// The data values inludes 17 bytes, which can be dynamically allocated as needed for each data field based on the size of the number

// Group Input mapping on robot appears as follows

// giKey1 : USINT;               giData1 : USINT;

// giKey2 : USINT;               giData2 : USINT;

// giKey3 : USINT;               giData3 : USINT;

// giKey4 : USINT;               giData4 : USINT;

// giKey5 : USINT;               giData5 : USINT;

// giKey6 : USINT;               giData6 : USINT;

// ...                           ...

// Example:

// Wall SAM ID is the first field of WallInfo step which is a large number 157864127 with needing 4 bytes to send.

// The next field of WallInfo is wall length which is 2000mm requiring 2 bytes to send.

// giKey1 is set to 4 and the number is divided into bytes occupying giData1,giData2,giData3, and giData4.

// giKey2 is set to 2 and the number is divided into bytes occupying giData5 and giData6.

// Function to pack NumbersToSend into bytes and determine key values

// first clear array

FOR i := 0 TO 14 DO
    Recipe_ByteQtyKey[i] := 0;
END_FOR

FOR i := 0 TO 16 DO
    Recipe_PackedBytes[i] := 0;
END_FOR

index := 0;

FOR i := 0 TO 10 DO

    // Determine how many bytes each number will occupy

    Recipe_ByteQtyKey[i] := 1;

    FOR j := 1 TO 3 DO
        IF ABS(RecipeData_ToSend[i]) > EXPT(2, (8 * j) - 1) THEN
            Recipe_ByteQtyKey[i] := INT_TO_USINT(j) + 1;

            // Make it easier to unpack by forcing data to be USINT (1), UINT (2) or UDINT (4)

            IF Recipe_ByteQtyKey[i] = 3 THEN
                Recipe_ByteQtyKey[i] := 4;
            END_IF
        END_IF
    END_FOR

    // Handle signed numbers

    numberToPack := RecipeData_ToSend[i];

    IF numberToPack < 0 THEN
        // Convert to Two's Complement for the required byte size

        CASE Recipe_ByteQtyKey[i] OF
            1:
                numberToPack := numberToPack AND 16#FF; // Mask for 8 bits
            2:
                numberToPack := numberToPack AND 16#FFFF; // Mask for 16 bits
            4:
                numberToPack := numberToPack AND 16#FFFFFFFF; // Mask for 32 bits
        END_CASE;
    END_IF

    // Now extract individual bytes from signed number

    IF Recipe_ByteQtyKey[i] = 1 THEN
        Recipe_PackedBytes[index] := UDINT_TO_USINT(numberToPack);
        index                     := index + 1;
    ELSE
        FOR j := Recipe_ByteQtyKey[i] - 1 TO 1 BY -1 DO
            Recipe_PackedBytes[index] := UDINT_TO_USINT(SHR(numberToPack, 8 * j));
            index                     := index + 1;
        END_FOR

        // Get the last byte

        Recipe_PackedBytes[index] := UDINT_TO_USINT(numberToPack);
        index                     := index + 1;
    END_IF

END_FOR;
END_METHOD

PROPERTY OtherInputs : ARRAY[0..7] OF USINT
GET
PUBLIC
VAR
END_VAR
OtherInputs := OtherInputsArray;
END_GET
END_PROPERTY

PROPERTY OtherOutputs : ARRAY[0..7] OF USINT
SET
PUBLIC
VAR
END_VAR
OtherOutputsArray := OtherOutputs;
END_SET
END_PROPERTY

END_FUNCTION_BLOCK

// Machine/Components/Safety/FB_Component_Safety
FUNCTION_BLOCK FB_Component_Safety EXTENDS FB_ComponentBase_SR
VAR_INPUT
    _SystemState : Tc3_PackML_V2.E_PMLState;
END_VAR

VAR_OUTPUT
END_VAR

VAR CONSTANT
    MAX_MGB_DOORS               : UDINT := 7;
    MAX_ESTOPS                  : UDINT := 8;
    MAX_LIGHT_CURTAINS          : UDINT := 4;
    MAX_AREA_SCANNERS           : UDINT := 3;
    COMPONENT_ALARM_COUNT       : UINT  := 9;
    MAX_PREPLATE_DOORS          : UDINT := 5;
    MAX_PREPLATE_LIGHT_CURTAINS : UDINT := 3;
END_VAR

VAR
    //Alarming
    ComponentAlarms : ARRAY[1..COMPONENT_ALARM_COUNT] OF FB_TcAlarm;

    // Component definitions here
    MGB_Door                      : ARRAY[1..MAX_MGB_DOORS] OF FB_Component_MGB_Door;
    E_Stop                        : ARRAY[1..MAX_ESTOPS] OF FB_DualChannelMonitor;
    E_Stop_Status                 : ARRAY[1..MAX_ESTOPS] OF ST_DualChannel_HMIStatus;
    Light_Curtains                : ARRAY[1..MAX_LIGHT_CURTAINS] OF FB_DualChannelMonitor;
    Light_Curtain_Status          : ARRAY[1..MAX_LIGHT_CURTAINS] OF ST_DualChannel_HMIStatus;
    Area_Scanners                 : ARRAY[1..MAX_AREA_SCANNERS] OF FB_DigitalSensor;
    Preplate_Doors                : ARRAY[1..MAX_PREPLATE_DOORS] OF FB_DualChannelMonitor;
    Preplate_Door_Status          : ARRAY[1..MAX_PREPLATE_DOORS] OF ST_DualChannel_HMIStatus;
    Light_Curtains_Preplate       : ARRAY[1..MAX_PREPLATE_LIGHT_CURTAINS] OF FB_DualChannelMonitor;
    Light_Curtain_Preplate_Status : ARRAY[1..MAX_PREPLATE_LIGHT_CURTAINS] OF ST_DualChannel_HMIStatus;

    FlashingLight : FB_PulseGenerator;

    SafetyRUN     AT %Q* : BOOL := TRUE;
    SafetyErrAckn AT %Q* : BOOL;
    SafetyReset   AT %Q* : BOOL;

    SafetyIsReset AT %I* : BOOL;
    SS1Input      AT %I* : BIT;
    SS1Output     AT %Q* : BIT;

    AirPressureOK AT %I* : BOOL;

    PrePlateAirPressureOK AT %I* : BOOL;

    OutfeedSafetyReset AT %Q* : BOOL;

    OutfeedSafetyIsReset AT %I* : BOOL;

    AutostopIsReset AT %I* : BOOL;

    OutfeedSafetyReset_Button3 AT %I* : BOOL;

    OutfeedSafetyReset_Button2 AT %I* : BOOL;

    OutfeedSafetyReset_HMI AT %I* : BOOL;

    SafetyStop AT %Q* : BOOL;

    SafetyOK_HMI_STATE : USINT;

    AutoStopOK_HMI_STATE : USINT;

    OutfeedAutoStopOK_HMI_STATE : USINT;

    SafetyOK_HMI_TEXT : STRING;

    AutoStopOK_HMI_TEXT : STRING;

    OutfeedAutoStopOK_HMI_TEXT : STRING;

    safetyState                   : USINT;
    tempSafetyOK_Main             : BOOL;
    tempSafetyCanBeReset_Main     : BOOL;
    tempSafetyReset_Main          : BOOL;
    tempSafetyOK_AutoStop         : BOOL;
    tempSafetyCanBeReset_AutoStop : BOOL;
    tempSafetyReset_AutoStop      : BOOL;
    tempSafetyOK_Outfeed          : BOOL;
    tempSafetyCanBeReset_Outfeed  : BOOL;
    tempSafetyReset_Outfeed       : BOOL;
    MainSafetyCanBeReset          : BOOL;
    AutoStopSafetyCanBeReset      : BOOL;
    OutfeedSafetyCanBeReset       : BOOL;
END_VAR

//! @summary This method serves as the entry point for all underlying FB logic
METHOD PUBLIC CyclicLogic

//! @description This method should be called cyclically by descendant function blocks by invoking <c>SUPER^.CyclicLogic()</c>.  Alternatively, the contents of this method could be reimplemented entirely in which case a call to this method would not be necessary.
// MGB_Door Names

MGB_Door[1].Name := 'Infeed';
MGB_Door[2].Name := 'Pre-Press';
MGB_Door[3].Name := 'Post_Press';
MGB_Door[4].Name := 'Assembly';
MGB_Door[5].Name := 'Jig_3 Door';
MGB_Door[6].Name := 'Jig_2 Door';
MGB_Door[7].Name := 'Preplate Cell'; // Button box and estop combined into "MGB Door" 

//Estop names
E_Stop[1].Name := 'MBI 1';
E_Stop[2].Name := 'MBI 1 Cable';
E_Stop[3].Name := 'MBI 2';
E_Stop[4].Name := 'MBI 2 Cable';
E_Stop[5].Name := 'HMI';
E_Stop[6].Name := 'Jig 3 Pendant';
E_Stop[7].Name := 'Jig 2 Pendant';
E_Stop[8].Name := 'Roof Truss Core';

//Outfeed Light curtain names
Light_Curtains[1].Name := 'Curtain 1';
Light_Curtains[2].Name := 'Curtain 2';
Light_Curtains[3].Name := 'Curtain 3';
Light_Curtains[4].Name := 'Curtain 4';

//Preplate Light curtain names
Light_Curtains_Preplate[1].Name := 'Curtain 1';
Light_Curtains_Preplate[2].Name := 'Curtain 2';
Light_Curtains_Preplate[3].Name := 'Curtain 3';

//Outfeed Light curtain names
Preplate_Doors[1].Name := 'Rack 1';
Preplate_Doors[2].Name := 'Rack 2';
Preplate_Doors[3].Name := 'Rack 3';
Preplate_Doors[4].Name := 'Rack 4';
Preplate_Doors[5].Name := 'Rack 5';

HMI_Status_Estops();
HMI_Status_LightCurtains();
HMI_Status_Preplate();

FOR i := 1 TO MAX_PREPLATE_DOORS DO
    Preplate_Doors[i].CyclicLogic();
    Preplate_Doors[i].InSimulation := _Simulate;
END_FOR

FOR i := 1 TO MAX_PREPLATE_LIGHT_CURTAINS DO
    Light_Curtains_Preplate[i].CyclicLogic();
    Light_Curtains_Preplate[i].InSimulation := _Simulate;
END_FOR

// Initialise Component

FlashingLight.OffTime := T#500MS;
FlashingLight.OnTime  := T#500MS;

FlashingLight.CyclicLogic();

MainSafetyCanBeReset := TRUE;

FOR i := 1 TO MAX_ESTOPS DO
    MainSafetyCanBeReset := MainSafetyCanBeReset AND E_Stop[i].BothChannelsOK;
END_FOR

FOR i := 1 TO MAX_MGB_DOORS DO
    MainSafetyCanBeReset := MainSafetyCanBeReset AND MGB_Door[i].Estop_CH_OK;
END_FOR

HMI_Indicators(Area             := 'Main',
               HMI_Text         := SafetyOK_HMI_TEXT,
               HMI_State        := SafetyOK_HMI_STATE,
               SafetyOK         := SafetyIsReset OR (_Simulate AND tempSafetyOK_Main),
               SafetyCanBeReset := MainSafetyCanBeReset,
               SafetyReset      := SafetyReset OR (tempSafetyReset_Main AND _Simulate));

IF MainSafetyCanBeReset AND _Simulate AND SafetyReset THEN
    tempSafetyOK_Main := TRUE;
ELSIF MainSafetyCanBeReset = FALSE THEN
    tempSafetyOK_Main := FALSE;
END_IF

AutoStopSafetyCanBeReset := TRUE;

FOR i := 1 TO MAX_MGB_DOORS - 2 DO
    AutoStopSafetyCanBeReset := AutoStopSafetyCanBeReset AND MGB_Door[i].AutoStop_CH_OK;
END_FOR

AutoStopSafetyCanBeReset := MainSafetyCanBeReset AND AutoStopSafetyCanBeReset;

HMI_Indicators(Area             := 'AutoStop',
               HMI_Text         := AutoStopOK_HMI_TEXT,
               HMI_State        := AutoStopOK_HMI_STATE,
               SafetyOK         := (AutostopIsReset AND SafetyIsReset) OR (_Simulate AND tempSafetyOK_AutoStop),
               SafetyCanBeReset := AutoStopSafetyCanBeReset,
               SafetyReset      := FALSE);

IF AutoStopSafetyCanBeReset AND _Simulate THEN
    tempSafetyOK_AutoStop := TRUE;
ELSIF AutoStopSafetyCanBeReset = FALSE THEN
    tempSafetyOK_AutoStop := FALSE;
END_IF

OutfeedSafetyCanBeReset := TRUE;

FOR i := 1 TO MAX_LIGHT_CURTAINS DO
    OutfeedSafetyCanBeReset := Light_Curtains[i].BothChannelsOK AND OutfeedSafetyCanBeReset;
END_FOR

OutfeedSafetyCanBeReset := MGB_Door[5].AutoStop_CH_OK AND OutfeedSafetyCanBeReset;
OutfeedSafetyCanBeReset := MGB_Door[6].AutoStop_CH_OK AND OutfeedSafetyCanBeReset;
OutfeedSafetyCanBeReset := MainSafetyCanBeReset AND OutfeedSafetyCanBeReset;

HMI_Indicators(Area             := 'Outfeed',
               HMI_Text         := OutfeedAutoStopOK_HMI_TEXT,
               HMI_State        := OutfeedAutoStopOK_HMI_STATE,
               SafetyOK         := (OutfeedSafetyIsReset AND SafetyIsReset) OR (_Simulate AND tempSafetyOK_Outfeed),
               SafetyCanBeReset := OutfeedSafetyCanBeReset,
               SafetyReset      := OutfeedSafetyReset OR (tempSafetyReset_Outfeed AND _Simulate));

IF OutfeedSafetyCanBeReset AND _Simulate AND OutfeedSafetyReset THEN
    tempSafetyOK_Outfeed := TRUE;
ELSIF OutfeedSafetyCanBeReset = FALSE THEN
    tempSafetyOK_Outfeed := FALSE;
END_IF

SS1Output := NOT SS1Input;

IF NOT _InitComplete THEN
    _InitComplete := Initialize();
    RETURN;
END_IF

IF SafetyReset THEN
    SafetyErrAckn := TRUE;
ELSE
    SafetyErrAckn := FALSE;
END_IF

OutfeedSafetyReset := OutfeedSafetyReset_Button3 OR OutfeedSafetyReset_Button2 OR OutfeedSafetyReset_HMI;

FOR i := 1 TO MAX_MGB_DOORS DO

    MGB_Door[i].CyclicLogic();
    MGB_Door[i].InSimulation := _Simulate;

    //Button lights and lock

    CASE _SystemState OF
        ePMLState_Idle:
            MGB_Door[i].Pause_LED.TurnOff();
            MGB_Door[i].Resume_LED.Flash();
            MGB_Door[i].Lock_Door.TurnOff();
        ePMLState_Holding, ePMLState_Suspending:
            MGB_Door[i].Pause_LED.Flash();
            MGB_Door[i].Resume_LED.TurnOff();
            MGB_Door[i].Lock_Door.TurnOn();
        ePMLState_Held, ePMLState_Suspended:
            MGB_Door[i].Pause_LED.TurnOff();
            MGB_Door[i].Resume_LED.TurnOn();
            MGB_Door[i].Lock_Door.TurnOff();
        ePMLState_Starting, ePMLState_Unholding, ePMLState_Unsuspending:
            MGB_Door[i].Pause_LED.TurnOff();
            MGB_Door[i].Resume_LED.Flash();
            MGB_Door[i].Lock_Door.TurnOn();
        ePMLState_Execute:
            MGB_Door[i].Pause_LED.TurnOn();
            MGB_Door[i].Resume_LED.TurnOff();
            MGB_Door[i].Lock_Door.TurnOn();
    ELSE
        MGB_Door[i].Pause_LED.TurnOff();
        MGB_Door[i].Resume_LED.TurnOff();
        MGB_Door[i].Lock_Door.TurnOff();
    END_CASE

    //estop light

    IF SafetyIsReset THEN
        MGB_Door[i].Estop_LED.TurnOff();
    ELSE
        IF MGB_Door[i].Estop_CH_OK THEN
            MGB_Door[i].Estop_LED.Flash();
        ELSE
            MGB_Door[i].Estop_LED.TurnOn();
        END_IF
        MGB_Door[i].Lock_Door.TurnOff();
    END_IF
    MGB_Door[i].SafetyReset := SafetyReset;
END_FOR

FOR i := 1 TO MAX_ESTOPS DO
    E_Stop[i].CyclicLogic();
    E_Stop[i].InSimulation := _Simulate;

    IF SafetyIsReset THEN
        E_Stop[i].LED.TurnOff();
    ELSE
        IF E_Stop[i].BothChannelsOK THEN
            E_Stop[i].LED.Flash();
        ELSE
            E_Stop[i].LED.TurnOn();
        END_IF
    END_IF
END_FOR

FOR i := 1 TO MAX_LIGHT_CURTAINS DO
    Light_Curtains[i].CyclicLogic();
    Light_Curtains[i].InSimulation := _Simulate;
END_FOR

SafetyStop := NOT (SafetyIsReset) OR NOT (AutostopIsReset);

SUPER^.CyclicLogic();
END_METHOD

(*! @summary Initializes event function blocks using this components's name*)
METHOD PROTECTED CreateEvents
F_CreateAllEventsInClass(Alarms     := ComponentAlarms,
                         ClassSize  := SIZEOF(TC_EVENTS.AMDTruss),
                         pInitEvent := ADR(TC_EVENTS.AMDTruss.InitReferenceEvent),
                         Prefix     := _Name);
END_METHOD

METHOD HMI_Indicators

VAR_INPUT
    Area             : STRING;
    HMI_Text         : REFERENCE TO STRING;
    HMI_State        : REFERENCE TO USINT;
    SafetyOK         : BOOL;
    SafetyCanBeReset : BOOL;
    SafetyReset      : BOOL;
END_VAR

VAR_INST
    Gif_TON       : TON;
    Safe_R_Trig_1 : R_TRIG;
    Safe_R_Trig_2 : R_TRIG;
END_VAR

Safe_R_Trig_1(CLK := SafetyOK);
Safe_R_Trig_2(CLK := SafetyReset);

IF Safe_R_Trig_1.Q THEN
    safetyState := 1;
END_IF

IF SafetyOK = FALSE THEN
    IF SafetyCanBeReset = FALSE THEN
        safetyState := 10;
    ELSE
        safetyState := 20;
    END_IF
END_IF

CASE safetyState OF
    1:
        HMI_Text  := CONCAT(Area, ' Safety OK');
        HMI_State := 1;
        Gif_TON(IN := FALSE);

        IF Safe_R_Trig_2.Q THEN
//             safetyState := 30;
        END_IF

    10:
        HMI_Text  := CONCAT(Area, ' Safety Not OK');
        HMI_State := 2;

    20:
        IF FlashingLight.PulseOutput THEN
            HMI_State := 3;
        ELSE
            HMI_State := 4;
        END_IF

        HMI_Text := CONCAT(Area, ' Safety Needs Reset');

    30:
        Gif_TON(IN := TRUE, PT := T#1S);

        IF Gif_TON.Q THEN
            safetyState := 1;
        END_IF

        HMI_Text  := CONCAT(Area, ' Safety Already Reset...');
        HMI_State := 5;

    99:
        ;
END_CASE
END_METHOD

METHOD HMI_Status_Estops
VAR_INPUT
END_VAR

VAR_INST
    EStop_R_TRIG    : ARRAY[1..MAX_ESTOPS] OF R_TRIG;
    EstopPressed    : ARRAY[1..MAX_ESTOPS] OF BOOL;
END_VAR
FOR i := 1 TO MAX_ESTOPS DO

    EStop_R_TRIG[i](CLK := NOT (E_Stop[i].BothChannelsOK));

    IF EStop_R_TRIG[i].Q THEN
        EstopPressed[i] := TRUE;
    END_IF

    IF SafetyReset THEN
        EstopPressed[i] := FALSE;
    END_IF

    E_Stop_Status[i].Name := E_Stop[i].Name;

    IF EstopPressed[i] THEN
        IF E_Stop[i].BothChannelsOK THEN
            E_Stop_Status[i].Status_Usint := 4;
            E_Stop_Status[i].Status_Str   := 'Reset Needed';
        ELSE
            E_Stop_Status[i].Status_Usint := 2;
            E_Stop_Status[i].Status_Str   := 'Estop Pressed';
        END_IF
    ELSE
        IF E_Stop[i].BothChannelsOK THEN
            E_Stop_Status[i].Status_Usint := 1;
            E_Stop_Status[i].Status_Str   := 'Estop OK';
        ELSE
            E_Stop_Status[i].Status_Usint := 2;
            E_Stop_Status[i].Status_Str   := 'Estop Pressed';
        END_IF
    END_IF
END_FOR
END_METHOD

METHOD HMI_Status_LightCurtains
VAR_INPUT
END_VAR

VAR_INST
    LC_R_TRIG    : ARRAY[1..MAX_ESTOPS] OF R_TRIG;
    LC_Tripped    : ARRAY[1..MAX_ESTOPS] OF BOOL;
END_VAR
FOR i := 1 TO MAX_LIGHT_CURTAINS DO

    LC_R_TRIG[i](CLK := NOT (Light_Curtains[i].BothChannelsOK));

    IF LC_R_TRIG[i].Q THEN
        LC_Tripped[i] := TRUE;
    END_IF

    IF OutfeedSafetyReset THEN
        LC_Tripped[i] := FALSE;
    END_IF

    Light_Curtain_Status[i].Name := Light_Curtains[i].Name;

    IF LC_Tripped[i] THEN
        IF Light_Curtains[i].BothChannelsOK THEN
            Light_Curtain_Status[i].Status_Usint := 4;
            Light_Curtain_Status[i].Status_Str   := 'Reset Needed';
        ELSE
            Light_Curtain_Status[i].Status_Usint := 2;
            Light_Curtain_Status[i].Status_Str   := 'Curtain Tripped';
        END_IF
    ELSE
        IF Light_Curtains[i].BothChannelsOK THEN
            Light_Curtain_Status[i].Status_Usint := 1;
            Light_Curtain_Status[i].Status_Str   := 'Curtain OK';
        ELSE
            Light_Curtain_Status[i].Status_Usint := 2;
            Light_Curtain_Status[i].Status_Str   := 'Curtain Tripped';
        END_IF
    END_IF
END_FOR
END_METHOD

METHOD HMI_Status_Preplate
VAR_INPUT
END_VAR
FOR i := 1 TO MAX_PREPLATE_DOORS DO
	Preplate_Door_Status[i].Name := Preplate_Doors[i].Name;
    IF Preplate_Doors[i].BothChannelsOK THEN
        Preplate_Door_Status[i].Status_Usint := 1;
        Preplate_Door_Status[i].Status_Str   := 'Door Closed';
    ELSE
        Preplate_Door_Status[i].Status_Usint := 2;
        Preplate_Door_Status[i].Status_Str   := 'Door Open';
    END_IF
END_FOR

FOR i := 1 TO MAX_PREPLATE_LIGHT_CURTAINS DO
	Light_Curtain_Preplate_Status[i].Name := Light_Curtains_Preplate[i].Name;
    IF Light_Curtains_Preplate[i].BothChannelsOK THEN
        Light_Curtain_Preplate_Status[i].Status_Usint := 1;
        Light_Curtain_Preplate_Status[i].Status_Str   := 'Curtain Clear';
    ELSE
        Light_Curtain_Preplate_Status[i].Status_Usint := 2;
        Light_Curtain_Preplate_Status[i].Status_Str   := 'Curtain Tripped';
    END_IF
END_FOR
END_METHOD

//! @summary Basic component initialization logic
METHOD PROTECTED Initialize : BOOL;

//! @description This method is called by <c>CyclicLogic()</c> as required
CreateEvents();

IF SUPER^.Initialize() THEN
    Initialize := TRUE;
END_IF
END_METHOD

(*! Provides basic error detection and event handling for this component*)
METHOD PROTECTED Monitoring
IF NOT AirPressureOK AND NOT ComponentAlarms[E_AMDTruss.LowAir].bRaised THEN
    RaiseAlarm2Args(ComponentAlarms[E_AMDTruss.LowAir], 'Air is low in the system', 'Please Turn on Air Before Continuing');
ELSIF AirPressureOK AND ComponentAlarms[E_AMDTruss.LowAir].bRaised THEN
    ComponentAlarms[E_AMDTruss.LowAir].Clear(0, 0);
END_IF

IF NOT SafetyIsReset AND NOT ComponentAlarms[E_AMDTruss.WarnMessage].bRaised THEN
    RaiseAlarm2Args(ComponentAlarms[E_AMDTruss.WarnMessage], 'Safety Reset Required', 'System Requires a Safety Reset to Continue');
ELSIF SafetyIsReset AND ComponentAlarms[E_AMDTruss.WarnMessage].bRaised THEN
    ComponentAlarms[E_AMDTruss.WarnMessage].Clear(0, 0);
END_IF

Super^.Monitoring();
END_METHOD

METHOD PauseInputs : BOOL
VAR_INPUT
END_VAR
PauseInputs := FALSE;

FOR i := 1 TO MAX_MGB_DOORS DO
    IF MGB_Door[i].Pause.Active THEN
        PauseInputs := TRUE;
        RETURN;
    END_IF
END_FOR
END_METHOD

METHOD ResumeInputs : BOOL
VAR_INPUT
END_VAR
ResumeInputs := FALSE;

FOR i := 1 TO MAX_MGB_DOORS DO
    IF MGB_Door[i].Resume.Active THEN
        ResumeInputs := TRUE;
        RETURN;
    END_IF
END_FOR
END_METHOD

PROPERTY AutostopOK : bool
GET
AutostopOK := AutostopIsReset OR _Simulate;
END_GET
END_PROPERTY

PROPERTY OutfeedAutostopOK : bool
GET
OutfeedAutostopOK := OutfeedSafetyIsReset OR _Simulate;
END_GET
END_PROPERTY

PROPERTY ParentResponseDefinitions : ARRAY[0..4] OF E_AlarmResponse
GET
ParentResponseDefinitions[TcEventSeverity.Verbose]  := E_AlarmResponse.NoResponse;
ParentResponseDefinitions[TcEventSeverity.Info]     := E_AlarmResponse.NoResponse;
ParentResponseDefinitions[TcEventSeverity.Warning]  := E_AlarmResponse.Suspend_Controlled;
ParentResponseDefinitions[TcEventSeverity.Error]    := E_AlarmResponse.Suspend_Controlled;
ParentResponseDefinitions[TcEventSeverity.Critical] := E_AlarmResponse.Suspend_Immediate;
END_GET
END_PROPERTY

PROPERTY SafetyOK : BOOL
GET
SafetyOK := SafetyIsReset OR _Simulate;
END_GET
END_PROPERTY

PROPERTY SystemState : Tc3_PackML_V2.E_PMLState
GET
SystemState := _SystemState;
END_GET
SET
_SystemState := SystemState;
END_SET
END_PROPERTY

END_FUNCTION_BLOCK

// Machine/Components/StackLight/Interfaces/I_StackLight
INTERFACE I_StackLight

PROPERTY SystemErrorPresent : BOOL
GET
END_GET
SET
END_SET
END_PROPERTY

END_INTERFACE

// Machine/Components/StackLight/FB_Component_Stacklight
FUNCTION_BLOCK FB_Component_StackLight EXTENDS FB_ComponentBase_SR IMPLEMENTS I_StackLight
VAR
    // Inputs

    _SystemState        : Tc3_PackML_V2.E_PMLState;
    _SystemErrorPresent : BOOL;

    // Outputs

    GreenLight : FB_Component_Indicator;
    AmberLight : FB_Component_Indicator;
    RedLight   : FB_Component_Indicator;
    Siren      : FB_Component_Indicator;

    // HMI

    // Alarms

    StackLightAlarms : ARRAY[1..STACKLIGHT_ALARMS_COUNT] OF FB_TcAlarm;

    // Internal variables

END_VAR

VAR CONSTANT
    STACKLIGHT_ALARMS_COUNT : UDINT := 5;
END_VAR

//! @summary This method serves as the entry point for all underlying FB logic
METHOD PUBLIC CyclicLogic

//! @description This method should be called cyclically by descendant function blocks by invoking <c>SUPER^.CyclicLogic()</c>.  Alternatively, the contents of this method could be reimplemented entirely in which case a call to this method would not be necessary.
// Initialise Component

IF NOT _InitComplete THEN
    _InitComplete := Initialize();
    RETURN;
END_IF

//// Main logic for StackLight control

CASE _SystemState OF
    ePMLState_Execute, ePMLState_Completing:
        IF NOT _SystemErrorPresent THEN
            GreenLight.TurnOn();
            AmberLight.TurnOff();
            RedLight.TurnOff();
            Siren.TurnOff();
        ELSE
            GreenLight.TurnOn();
            AmberLight.TurnOff();
            RedLight.Flash();
            Siren.TurnOff();
        END_IF

    ePMLState_Idle:
        GreenLight.Flash();
        AmberLight.TurnOff();
        RedLight.TurnOff();
        Siren.TurnOff();

    ePMLState_Starting, ePMLState_Unholding, ePMLState_Unsuspending:
        GreenLight.TurnOn();
        AmberLight.TurnOff();
        RedLight.TurnOff();
        Siren.OffTime := TIME#500MS;
        Siren.Flash();

    ePMLState_Holding:
        GreenLight.TurnOff();
        AmberLight.Flash();
        RedLight.TurnOff();
        Siren.TurnOff();

    ePMLState_Held:
        GreenLight.TurnOff();
        AmberLight.TurnOn();
        RedLight.TurnOff();
        Siren.TurnOff();

    ePMLState_Suspended:
        GreenLight.TurnOff();
        AmberLight.TurnOn();
        RedLight.Flash();
        Siren.OffTime := TIME#5S;
        Siren.Flash();

    ePMLState_Stopped, ePMLState_Clearing, ePMLState_Aborted, ePMLState_Aborting, ePMLState_Complete:
        GreenLight.TurnOff();
        AmberLight.TurnOff();
        RedLight.TurnOn();
        Siren.TurnOff();

    ePMLState_Resetting:
        GreenLight.TurnOff();
        AmberLight.TurnOff();
        RedLight.Flash();
        Siren.TurnOn();

ELSE
    GreenLight.TurnOff();
    AmberLight.TurnOff();
    RedLight.TurnOff();
    Siren.TurnOff();
END_CASE

IF _SystemErrorPresent THEN
    RedLight.Flash();
    Siren.OnTime  := T#100MS;
    Siren.OffTime := T#10S;
    Siren.Flash();
END_IF

GreenLight.CyclicLogic();
AmberLight.CyclicLogic();
RedLight.CyclicLogic();
Siren.CyclicLogic();

// Component Error

//{error 'Create Component has Error'}

//_Error := TRUE;

//_ErrorID := 9999;

// Component Busy

//{error 'Create Component is Busy'}

IF TRUE THEN
    _Busy := TRUE;
ELSE
    _Busy := FALSE;
END_IF

// Call Super

SUPER^.CyclicLogic();

// Set Current Alarm Severity

////_CurrentAlarmSeverity := F_GetMaxSeverityRaised(Alarms := StackLightAlarms, CurrentSeverity := _CurrentSeverity, Severity := _CurrentAlarmSeverity);
END_METHOD

METHOD PROTECTED CreateEvents
VAR_INPUT
END_VAR
SUPER^.CreateEvents();
END_METHOD

//! @summary Basic component initialization logic
METHOD PROTECTED Initialize : BOOL;

//! @description This method is called by <c>CyclicLogic()</c> as required
CreateEvents();

IF SUPER^.Initialize() THEN
    Initialize := TRUE;
END_IF
END_METHOD

METHOD PROTECTED Monitoring
VAR_INPUT
END_VAR
SUPER^.Monitoring();
END_METHOD

PROPERTY SystemErrorPresent : BOOL
GET
SystemErrorPresent := _SystemErrorPresent;
END_GET
SET
_SystemErrorPresent := SystemErrorPresent;
END_SET
END_PROPERTY

PROPERTY SystemState : Tc3_PackML_V2.E_PMLState
GET
SystemState := _SystemState;
END_GET
SET
_SystemState := SystemState;
END_SET
END_PROPERTY

END_FUNCTION_BLOCK

// Machine/Components/StackLight_MBI/Interfaces/I_StackLight_1
INTERFACE I_StackLight_1

PROPERTY MyInput : BOOL
GET
END_GET
SET
END_SET
END_PROPERTY

PROPERTY MyOutput : E_PMLState
GET
END_GET
SET
END_SET
END_PROPERTY

END_INTERFACE

// Machine/Components/StackLight_MBI/FB_Component_Stacklight_MBI
FUNCTION_BLOCK FB_Component_Stacklight_MBI EXTENDS FB_ComponentBase_SR
VAR
    // Inputs

    _SystemState        : Tc3_PackML_V2.E_PMLState;
    _SystemErrorPresent : BOOL;

    // Outputs

    WhiteLight : FB_Component_Indicator;
    AmberLight : FB_Component_Indicator;
    Siren      : FB_Component_Indicator;

    // HMI

    // Alarms

    StackLightAlarms : ARRAY[1..STACKLIGHT_ALARMS_COUNT] OF FB_TcAlarm;

    // Internal variables

END_VAR

VAR CONSTANT
    STACKLIGHT_ALARMS_COUNT : UDINT := 5;
END_VAR

//! @summary This method serves as the entry point for all underlying FB logic
METHOD PUBLIC CyclicLogic

//! @description This method should be called cyclically by descendant function blocks by invoking <c>SUPER^.CyclicLogic()</c>.  Alternatively, the contents of this method could be reimplemented entirely in which case a call to this method would not be necessary.
// Initialise Component

IF NOT _InitComplete THEN
    _InitComplete := Initialize();
    RETURN;
END_IF

WhiteLight.CyclicLogic();
AmberLight.CyclicLogic();
Siren.CyclicLogic();

// Component Error

//{error 'Create Component has Error'}

//_Error := TRUE;

//_ErrorID := 9999;

// Component Busy

//{error 'Create Component is Busy'}

IF TRUE THEN
    _Busy := TRUE;
ELSE
    _Busy := FALSE;
END_IF

// Call Super

SUPER^.CyclicLogic();

// Set Current Alarm Severity

////_CurrentAlarmSeverity := F_GetMaxSeverityRaised(Alarms := StackLightAlarms, CurrentSeverity := _CurrentSeverity, Severity := _CurrentAlarmSeverity);
END_METHOD

METHOD PROTECTED CreateEvents
VAR_INPUT
END_VAR
SUPER^.CreateEvents();
END_METHOD

//! @summary Basic component initialization logic
METHOD PROTECTED Initialize : BOOL;

//! @description This method is called by <c>CyclicLogic()</c> as required
CreateEvents();

IF SUPER^.Initialize() THEN
    Initialize := TRUE;
END_IF
END_METHOD

METHOD PROTECTED Monitoring
VAR_INPUT
END_VAR
SUPER^.Monitoring();
END_METHOD

PROPERTY MyOutput : Tc3_PackML_V2.E_PMLState
GET
MyOutput := _SystemState;
END_GET
SET
_SystemState := MyOutput;
END_SET
END_PROPERTY

PROPERTY SystemErrorPresent : BOOL
GET
SystemErrorPresent := _SystemErrorPresent;
END_GET
SET
_SystemErrorPresent := SystemErrorPresent;
END_SET
END_PROPERTY

END_FUNCTION_BLOCK

// Machine/Components/Template_MyComponent/Interfaces/I_MyComponent
INTERFACE I_MyComponent

PROPERTY SystemErrorPresent : BOOL
GET
END_GET
SET
END_SET
END_PROPERTY

PROPERTY SystemState : E_PMLState
GET
END_GET
SET
END_SET
END_PROPERTY

END_INTERFACE

// Machine/Components/Template_MyComponent/FB_Component_MyComponent
FUNCTION_BLOCK FB_Component_MyComponent EXTENDS FB_ComponentBase_SR IMPLEMENTS I_MyComponent
VAR
    // Inputs

    MyInput AT %I* : BOOL;

    // Outputs

    MyOutput AT %Q* : BOOL;

    // HMI

    MyComponent_HMI : ST_ComponentMyComponent_HMI;

    // Alarms

    MyComponentAlarms : ARRAY[1..MY_COMPONENT_ALARMS_COUNT] OF FB_TcAlarm;

    // Internal variables

    _MyVarProperty1 : BOOL;
    _MyVarProperty2 : BOOL;
    MyVarEnternal1  : BOOL;
    MyVarEnternal2  : BOOL;

END_VAR

VAR CONSTANT
    MY_COMPONENT_ALARMS_COUNT : UDINT := 5;
END_VAR

//! @summary This method serves as the entry point for all underlying FB logic
METHOD PUBLIC CyclicLogic

//! @description This method should be called cyclically by descendant function blocks by invoking <c>SUPER^.CyclicLogic()</c>.  Alternatively, the contents of this method could be reimplemented entirely in which case a call to this method would not be necessary.
// Initialise Component

IF NOT _InitComplete THEN
    _InitComplete := Initialize();
    RETURN;
END_IF

//Custom Component Logic goes here

// Call Super

SUPER^.CyclicLogic();

// Set Current Alarm Severity

_CurrentAlarmSeverity := F_GetMaxSeverityRaised(Alarms := MyComponentAlarms, CurrentSeverity := _CurrentAlarmSeverity);
END_METHOD

METHOD PROTECTED CreateEvents
VAR_INPUT
END_VAR
SUPER^.CreateEvents();
END_METHOD

//! @summary Basic component initialization logic
METHOD PROTECTED Initialize : BOOL;

//! @description This method is called by <c>CyclicLogic()</c> as required
CreateEvents();

IF SUPER^.Initialize() THEN
    Initialize := TRUE;
END_IF
END_METHOD

METHOD PROTECTED Monitoring
VAR_INPUT
END_VAR
SUPER^.Monitoring();
END_METHOD

PROPERTY MyInput : BOOL
GET
MyInput := _Present;
END_GET
SET
_Present := MyInput;
END_SET
END_PROPERTY

PROPERTY MyOutput : BOOL
GET
MyOutput := _MyOutput;
END_GET
SET
_SystemState := MyOutput;
END_SET
END_PROPERTY

END_FUNCTION_BLOCK

// Machine/Components/VFD/Interfaces/I_VFD
INTERFACE I_VFD

METHOD Jog : BOOL
VAR_INPUT
    JogFW : BOOL := FALSE;
    JogBW : BOOL := FALSE;
END_VAR
END_METHOD

METHOD Stop : BOOL
VAR_INPUT
END_VAR
END_METHOD

END_INTERFACE

// Machine/Components/VFD/FB_Component_ABB_VFD_EC
FUNCTION_BLOCK FB_Component_ABB_VFD_EC EXTENDS FB_ComponentBase IMPLEMENTS I_VFD
VAR_INPUT
END_VAR

VAR_OUTPUT
END_VAR

VAR

    //ABB	: AXIS_Ref;
    ABB_State : INT;
    AbsVel    : INT := 1200;
    DirPos    : INT := -1;
    DirNeg    : INT := 1;

    // ABB Drive StatusWord
    ABBSW           AT %I* : UINT;
    ReadySwOn       AT %I* : BOOL;
    SwitchedOn      AT %I* : BOOL;
    OpEnabled       AT %I* : BOOL;
    Fault           AT %I* : BOOL;
    VoltageEnable   AT %I* : BOOL;
    QuickStopActive AT %I* : BOOL;
    SwitchOnDisable AT %I* : BOOL;
    Warning         AT %I* : BOOL;
    AtSetpoint      AT %I* : BOOL;
    Remote          AT %I* : BOOL;
    InternalLimit   AT %I* : BOOL;

    // ABB Drive ControlWord
    ABBCW         AT %Q* : UINT;
    Vel           AT %Q* : INT;
    SwitchOn      AT %Q* : BOOL;
    EnableVoltage AT %Q* : BOOL;
    QuickStop     AT %Q* : BOOL;
    EnableOp      AT %Q* : BOOL;
    RampOut       AT %Q* : BOOL;
    RampHold      AT %Q* : BOOL;
    RampIn        AT %Q* : BOOL;
    bReset        AT %Q* : BOOL;
    RemoteCmd     AT %Q* : BOOL;
    ExtCntrl      AT %Q* : BOOL;

    //Motion Command and Limit Switches
    DriveSW AT %I* : UINT;
    DriveCW AT %Q* : UINT;

    LimitSwitchExt AT %I* : BOOL;
    LimitSwitchRet AT %I* : BOOL;

    _Extended  : BOOL;
    _Retracted : BOOL;
END_VAR

METHOD CyclicLogic
ABBCW.0  := SwitchOn;
ABBCW.1  := EnableVoltage;
ABBCW.2  := QuickStop;
ABBCW.3  := EnableOp;
ABBCW.4  := RampOut;
ABBCW.5  := RampHold;
ABBCW.6  := RampIn;
ABBCW.7  := bReset;
ABBCW.10 := RemoteCmd;
ABBCW.11 := ExtCntrl;

ReadySwOn       := ABBSW.0;
SwitchedOn      := ABBSW.1;
OpEnabled       := ABBSW.2;
Fault           := ABBSW.3;
VoltageEnable   := ABBSW.4;
QuickStopActive := ABBSW.5;
SwitchOnDisable := ABBSW.6;
Warning         := ABBSW.7;
AtSetpoint      := ABBSW.8;
Remote          := ABBSW.9;
InternalLimit   := ABBSW.11;

LimitSwitchExt := DriveSW.0;
LimitSwitchRet := DriveSW.1;

_Extended  := NOT LimitSwitchExt;
_Retracted := NOT LimitSwitchRet;

IF (ReadySwOn = FALSE OR Fault = 1) AND ABB_State = 3 THEN
    ABB_State := 0;
END_IF

//ABB DRIVE COMMUNICATION PROFILE STATE MACHINE
CASE ABB_State OF

    //CHECK THAT DEVICE IS IN REMOTE
    0:
        bReset := 0;

        IF Remote AND Fault = 0 THEN
            ABB_State := 1;
        END_IF

        //NOT READY TO SWITCH ON
    1:
        SwitchOn      := 0;
        EnableVoltage := 1;
        QuickStop     := 1;

        IF ReadySwOn AND SwitchedOn = FALSE THEN
            ABB_State := 2;
        END_IF

        //READY TO SWITCH ON
    2:
        SwitchOn := 1;

        IF SwitchedOn THEN
            ABB_State := 3;
        END_IF

        // OPERATION ENABLED
    3:

        //SWITCH ON DISABLED
    5:
        ;

        //FAULT
    6:
        SwitchOn      := 0;
        bReset        := 1;
        ABB_State     := 0;
        EnableVoltage := 0;
        QuickStop     := 0;

END_CASE

SUPER^.CyclicLogic();
END_METHOD

PROPERTY Extended : BOOL
GET
Extended := _Extended;
END_GET
END_PROPERTY

PROPERTY Retracted : BOOL
GET
Retracted := _Retracted;
END_GET
END_PROPERTY

METHOD Jog : BOOL
VAR_INPUT
    JogFW : BOOL := FALSE;
    JogBW : BOOL := FALSE;
END_VAR
IF ABB_State = 3 THEN
    IF JogFW AND LimitSwitchExt THEN //EXTEND UNTIL LIMIT SWITCH
        EnableOp := 1;
        RampOut  := 1;
        RampHold := 1;
        RampIn   := 1;
        Vel      := DirPos * AbsVel;
    ELSIF JogBW AND LimitSwitchRet THEN //RETRACT UNTIL LIMIT SWITCH
        EnableOp := 1;
        RampOut  := 1;
        RampHold := 1;
        RampIn   := 1;
        Vel      := DirNeg * AbsVel;
    ELSIF NOT LimitSwitchExt THEN //DISABLE WHEN POSITIVE LIMIT SWITCH IS TRIGGERED
        JogFW    := FALSE;
        EnableOp := 0;
        RampOut  := 0;
    ELSIF NOT LimitSwitchRet THEN //DISABLE WHEN NEGATIVE LIMIT SWITCH IS TRIGGERED
        JogBW    := FALSE;
        EnableOp := 0;
        RampOut  := 0;
    ELSE //DISABLE WHEN SIGNALS TO BOTH LIMIT SWITCHES ARE INTERRUPTED
        EnableOp := 0;
        RampOut  := 0;
    END_IF
END_IF
END_METHOD

METHOD Reset : BOOL
IF SUPER^.Reset() THEN
    IF Fault THEN
        bReset := TRUE;
    ELSE
        Reset  := TRUE;
        bReset := FALSE;
    END_IF
END_IF
END_METHOD

METHOD Stop : BOOL
EnableOp := 0;
RampOut  := 0;
END_METHOD

END_FUNCTION_BLOCK

// Machine/Components/VFD/FB_Component_ABB_VFD_EIP
FUNCTION_BLOCK FB_Component_ABB_VFD_EIP EXTENDS FB_ComponentBase_SR IMPLEMENTS I_VFD
VAR

    // Outputs
    _ControlWord  AT %Q* : UDINT;
    _EnableMotor  AT %Q* : BOOL;
    _FaultReset   AT %Q* : BOOL;
    _Frequency    AT %Q* : WORD;
    _JogFwd       AT %Q* : BOOL;
    _JogRvs       AT %Q* : BOOL;
    _ReferenceVel AT %Q* : INT;

    // Inputs
    _StatusWord   AT %I* : UDINT;
    _Enabled      AT %I* : BOOL;
    _CommandedVel AT %I* : INT;
    _Faulted      AT %I* : BOOL;
    _Warning      AT %I* : BOOL;
    _FwdActive    AT %I* : BOOL;
    _RvsActive    AT %I* : BOOL;
    _AtSpeed      AT %I* : BOOL;
    _State        AT %I* : USINT;
    // Alarms

    IndicatorAlarms : ARRAY[1..Indicator_ALARMS_COUNT] OF FB_TcAlarm;

    // Internal variables

    Pulse : FB_PulseGenerator;

END_VAR

VAR CONSTANT
    Indicator_ALARMS_COUNT : UDINT := 5;
END_VAR

//! @summary This method serves as the entry point for all underlying FB logic
METHOD PUBLIC CyclicLogic

//! @description This method should be called cyclically by descendant function blocks by invoking <c>SUPER^.CyclicLogic()</c>.  Alternatively, the contents of this method could be reimplemented entirely in which case a call to this method would not be necessary.
// Initialise Component

IF NOT _InitComplete THEN
    _InitComplete := Initialize();
    RETURN;
END_IF

// Call Super

SUPER^.CyclicLogic();

// Set Current Alarm Severity

_CurrentAlarmSeverity := F_GetMaxSeverityRaised(Alarms := IndicatorAlarms, CurrentSeverity := _CurrentAlarmSeverity);
END_METHOD

METHOD Disable : BOOL
VAR_INPUT
END_VAR
Disable := FALSE;
JogFwd  := FALSE;
JogRvs  := FALSE;

IF FwdActive = FALSE AND RvsActive = FALSE THEN
    Disable := TRUE;
END_IF
END_METHOD

METHOD Enable : BOOL
VAR_INPUT
END_VAR
Enable := FALSE;

IF Enabled = TRUE THEN
    Enable := TRUE;
END_IF
END_METHOD

//! @summary Basic component initialization logic
METHOD PROTECTED Initialize : BOOL;

//! @description This method is called by <c>CyclicLogic()</c> as required
CreateEvents();

IF SUPER^.Initialize() THEN
    Initialize := TRUE;
END_IF
END_METHOD

METHOD Jog : BOOL
VAR_INPUT
    JogFW : BOOL := FALSE;
    JogBW : BOOL := FALSE;
END_VAR
IF JogFW THEN
    Jog    := FALSE;
    JogFwd := TRUE;
    JogRvs := FALSE;

    IF FwdActive AND AtSpeed THEN
        Jog := TRUE;
    END_IF
ELSIF JogBW THEN

    Jog    := FALSE;
    JogFwd := FALSE;
    JogRvs := TRUE;

    IF RvsActive AND AtSpeed THEN
        Jog := TRUE;
    END_IF

END_IF
END_METHOD

METHOD PROTECTED Monitoring
VAR_INPUT
END_VAR
SUPER^.Monitoring();
END_METHOD

METHOD Reset : BOOL
Reset := FALSE;

IF Faulted THEN
    FaultReset := TRUE;
ELSE
    FaultReset := FALSE;
    Reset      := TRUE;
END_IF
END_METHOD

METHOD Stop : BOOL
VAR_INPUT
END_VAR
Stop   := FALSE;
JogFwd := FALSE;
JogRvs := FALSE;

IF FwdActive = FALSE AND RvsActive = FALSE THEN
    Stop := TRUE;
END_IF
END_METHOD

PROPERTY AtSpeed : bool
GET
AtSpeed := _AtSpeed;
END_GET
END_PROPERTY

PROPERTY CommandedVel : WORD
GET
CommandedVel := INT_TO_WORD(_CommandedVel);
END_GET
END_PROPERTY

PROPERTY Enabled : bool
GET
Enabled := _Enabled;
END_GET
END_PROPERTY

PROPERTY Faulted : bool
GET
Faulted := _Faulted;
END_GET
END_PROPERTY

PROPERTY FaultReset : bool
SET
_FaultReset := FaultReset;
END_SET
END_PROPERTY

PROPERTY Frequency : WORD
SET
_Frequency := Frequency;
END_SET
END_PROPERTY

PROPERTY FwdActive : bool
GET
FwdActive := _FwdActive;
END_GET
END_PROPERTY

PROPERTY JogFwd : bool
SET
_JogFwd := JogFwd;
END_SET
END_PROPERTY

PROPERTY JogRvs : bool
SET
_JogRvs := JogRvs;
END_SET
END_PROPERTY

PROPERTY ReferenceVel : WORD
SET
_ReferenceVel := WORD_TO_INT(ReferenceVel);
END_SET
END_PROPERTY

PROPERTY RvsActive : bool
GET
RvsActive := _RvsActive;
END_GET
END_PROPERTY

PROPERTY State : USINT
GET
State := _State;
END_GET
END_PROPERTY

PROPERTY Warning : bool
GET
Warning := _Warning;
END_GET
END_PROPERTY

END_FUNCTION_BLOCK

// Machine/EquipmentModules/EquipmentModule_SR/Interfaces/I_CommandStepParser
INTERFACE I_CommandStepParser

METHOD AssemblyEndParse : BOOL

VAR_INPUT
    Step          : ST_CSV_Step;
    StepDetailOut : REFERENCE TO ST_AssemblyEnd;
END_VAR
END_METHOD

METHOD AssemblyStartParse : BOOL
VAR_INPUT
    Step    : ST_CSV_Step;
    StepOut : REFERENCE TO ST_AssemblyStart;
END_VAR
END_METHOD

METHOD BoardInfoParse : BOOL
VAR_INPUT
    Step    : ST_CSV_Step;
    StepOut : REFERENCE TO ST_BoardInfo;
END_VAR
END_METHOD

METHOD BoardParse : BOOL
VAR_INPUT
    Step    : ST_CSV_Step;
    StepOut : REFERENCE TO ST_Board;
END_VAR
END_METHOD

METHOD NailPlateParse : BOOL
VAR_INPUT
    Step    : ST_CSV_Step;
    StepOut : REFERENCE TO ST_BoardInfo;
END_VAR
END_METHOD

METHOD TrussInfoParse : BOOL
VAR_INPUT
    Step    : ST_CSV_Step;
    StepOut : REFERENCE TO ST_TrussInfo;
END_VAR
END_METHOD

END_INTERFACE

// Machine/EquipmentModules/EquipmentModule_SR/Interfaces/I_CommandSteps
INTERFACE I_CommandSteps

METHOD AssemblyEnd : BOOL
VAR_INPUT
END_VAR
END_METHOD

METHOD AssemblyStart : BOOL
VAR_INPUT
END_VAR
END_METHOD

METHOD Board : BOOL
VAR_INPUT
END_VAR
END_METHOD

METHOD BoardInfo : BOOL
VAR_INPUT
END_VAR
END_METHOD

METHOD NailPlate : BOOL
VAR_INPUT
END_VAR
END_METHOD

METHOD TrussInfo : BOOL
VAR_INPUT
END_VAR
END_METHOD

END_INTERFACE

// Machine/EquipmentModules/EquipmentModule_SR/Interfaces/I_EquipmentModule_SR
INTERFACE I_EquipmentModule_SR EXTENDS I_PackML_BaseModule

PROPERTY EquipmentModuleID : E_EM_Index;
GET
END_GET
SET
END_SET
END_PROPERTY

PROPERTY InSimulation : BOOL
SET
END_SET
END_PROPERTY

PROPERTY SafetyOK : BOOL
SET
END_SET
END_PROPERTY

METHOD SimulationOff : BOOL
VAR_INPUT
END_VAR
END_METHOD

METHOD SimulationOn : BOOL
VAR_INPUT
END_VAR
END_METHOD

END_INTERFACE

// Machine/EquipmentModules/EquipmentModule_SR/Interfaces/I_MachineComms
INTERFACE I_MachineComms extends I_PackML_BaseModule

PROPERTY Step : DINT
SET
END_SET
END_PROPERTY

PROPERTY WaitSync : E_WaitSync
GET
END_GET
SET
END_SET
END_PROPERTY

END_INTERFACE

// Machine/EquipmentModules/EquipmentModule_SR/FB_EquipmentModule_SR
FUNCTION_BLOCK FB_EquipmentModule_SR EXTENDS FB_PackML_BaseModule IMPLEMENTS I_EquipmentModule_SR
VAR

    EquipmentModule_Alarms : ARRAY[1..Global.MAX_ALARM_COUNT] OF FB_TcAlarm;

    ipSubmodules_SR : ARRAY[1..Parameters_PackML_Base.MAX_NO_OF_SUBMODULES] OF I_EquipmentModule_SR := [];

    //HMI Control for EM

    fbControlSourceHMI : FB_ControlSource_HMI;

    ErrorInput : BOOL;
    WarnInput  : BOOL;
    InfoInput  : BOOL;

    //WaitSync varables

    _ResponseWaitSync  : E_WaitSync;
    _RequestedWaitSync : E_WaitSync;
    _Handshake_State   : DINT;
    _Step              : DINT;

    //Iterator step

    _CurrentStep  : DINT := 1;
    _TaskState    : E_TaskState;
    LastStepRan   : DINT; // Current step number
    _StepToRun    : DINT := 1;
    _InSimulation : BOOL;
    _SafetyOK     : BOOL;
    //Motor Resetting

    _MotorHoming       : BOOL := TRUE;
    _MotorsReset       : BOOL;
    _MotorsInitialized : BOOL;
    _MotorsHomed       : BOOL;
    _MotorResetState   : DINT;
    _MotorInitState    : DINT;
    _MotorHomeState    : DINT;
    _AlignNeeded       : BOOL;
    _AlignGearInState  : DINT;

    _RecoverBoardNum : DINT;

    _EquipmentModuleID : E_EM_Index;

    _CurrentCommandName : STRING;

    _SubmodulesReset : BOOL;
    _ComponentsReset : BOOL;
    i                : UDINT;
    j                : UDINT;
    k                : UDINT;
    ParseDone        : BOOL;

    testbool   : BOOL;
    testbool1  : BOOL;
    testbool2  : BOOL;
    testbool3  : BOOL;
    testbool4  : BOOL;
    testbool5  : BOOL;
    testbool6  : BOOL;
    testbool7  : BOOL;
    testbool8  : BOOL;
    testbool9  : BOOL;
    testbool10 : BOOL;
    testbool11 : BOOL;

    testmessagebox1 : BOOL;
    testmessagebox2 : BOOL;
    testmessagebox3 : BOOL;

    teststring : STRING;
    testlreal  : LREAL;
	tcMessage: Tc3_Database.I_TcMessage;
	
END_VAR

VAR
    MessageBox_Data     : ST_MessageBox_Data;
    MessageBox_Response : ST_MessageBox_Response;

    AutoUnsuspendCheck_TON : TON;
    AutoUnsuspendReset_TON : TON;
    AutoUnsuspendAvailable : BOOL;

    _ForceHold : BOOL;

	HMI_INPUT : ARRAY[1..20] OF BOOL;
	HMI_OUTPUT : ARRAY[1..20] OF BOOL;
	HMI_R_TRIG : ARRAY[1..50] OF R_TRIG;
END_VAR

VAR
	//data logging
    nState : INT;

    //for generating timestamp
    fbGetSystemTime1 : GetSystemTime;
    dwTimeLoDW       : DWORD;
    dwTimeHiDW       : DWORD;
    tFileTime        : T_FILETIME;
    nTimestamp       : LINT;

    //for creating table
    fbPLCDBCreate : FB_PLCDBCreateEvt(sNetID := '', tTimeout := T#5S);
    aTblCfg       : ARRAY[0..3] OF ST_ColumnInfo;

    //for insert samples
    fbPLCDBCmd : FB_PLCDBCmdEvt(sNetID := '', tTimeout := T#19S);
    aPara      : ARRAY[0..3] OF ST_ExpParameter;
    sCmd1      : STRING(255);
    sCmd2      : STRING(255);
    sCmd       : STRING(512); //CONCAT of sCmd1 and sCmd2

    //Data buffer
    aWriteSQL : ARRAY[0..19] OF BOOL;
    stData    : ARRAY[0..19, 0..99] OF ST_EquipmentModuleLog;

    //buffer index
    nWriteBufferIndex : INT := 0;
    nWriteIndex       : INT := 0;
    nSQLIndex         : INT := 0;

    fbGetSystemTime : GETSYSTEMTIME;
    fileTime        : T_FILETIME;
    dtTime          : DATE_AND_TIME;
END_VAR

METHOD AssemblyEndParse : BOOL
VAR_INPUT
    Step          : ST_CSV_Step;
    StepDetailOut : REFERENCE TO ST_AssemblyEnd;
END_VAR
StepDetailOut.SeqID := Step.seqID;

AssemblyEndParse := TRUE;
END_METHOD

METHOD AssemblyStartParse : BOOL
VAR_INPUT
    Step    : ST_CSV_Step;
    StepOut : REFERENCE TO ST_AssemblyStart;
END_VAR
StepOut.ComponentID := Step.Details[1].Datas[1];

AssemblyStartParse := TRUE;
END_METHOD

METHOD BoardInfoParse : BOOL
VAR_INPUT
    Step    : ST_CSV_Step;
    StepOut : REFERENCE TO ST_BoardInfo;
END_VAR

VAR
    Detail          : ST_CSV_Detail;
    conversionError : BOOL := FALSE;
END_VAR
// Ensure there's at least one detail in the step
IF Step.DetailCount < 1 THEN
    BoardInfoParse := FALSE;
    RETURN;
END_IF

// Use the first detail
Detail := Step.Details[1];

// Check if the detail has enough data fields (we need at least 6 fields)
IF Detail.DataCount < 6 THEN
    BoardInfoParse := FALSE;
    RETURN;
END_IF

// BoardID
StepOut.BoardID := Detail.Datas[1];

// BoardNumber
StepOut.BoardNumber := STRING_TO_INT(Detail.Datas[2]);

// BoardWidth
StepOut.BoardWidth := STRING_TO_REAL(Detail.Datas[3]);

// BoardHeight
StepOut.BoardHeight := STRING_TO_REAL(Detail.Datas[4]);

// BoardLength
StepOut.BoardLength := STRING_TO_REAL(Detail.Datas[5]);

// TotalPlates
StepOut.TotalPlates := STRING_TO_INT(Detail.Datas[6]);

BoardInfoParse := TRUE;
END_METHOD

METHOD BoardParse : BOOL
VAR_INPUT
    Step    : ST_CSV_Step;
    StepOut : REFERENCE TO ST_Board;
END_VAR

// For simplicity, we'll use the first detail
VAR
    Detail : ST_CSV_Detail;
END_VAR
// Ensure there's at least one detail in the step
IF Step.DetailCount < 1 THEN
    BoardParse := FALSE;
    RETURN;
END_IF

Detail := Step.Details[1];

// Check if the detail has enough data fields
IF Detail.DataCount < 7 THEN
    BoardParse := FALSE;
    RETURN;
END_IF

// BoardID
StepOut.BoardID := Detail.Datas[1];

// BoardWidth
StepOut.BoardWidth := STRING_TO_REAL(Detail.Datas[2]);

// BoardHeight
StepOut.BoardHeight := STRING_TO_REAL(Detail.Datas[3]);

// BoardLength
StepOut.BoardLength := STRING_TO_REAL(Detail.Datas[4]);

// BoardNumber
StepOut.BoardNumber := STRING_TO_INT(Detail.Datas[5]);

// LeadingEdgeBevelOffset
StepOut.LeadingEdgeBevelOffset := STRING_TO_REAL(Detail.Datas[6]);

// TrailingEdgeBevelOffset
StepOut.TrailingEdgeBevelOffset := STRING_TO_REAL(Detail.Datas[7]);

BoardParse := TRUE;
END_METHOD

METHOD IndexConveyorParse : BOOL
VAR_INPUT
    Step    : ST_CSV_Step;
    StepOut : REFERENCE TO ST_IndexConveyor;
END_VAR

VAR
    Detail          : ST_CSV_Detail;
    conversionError : BOOL := FALSE;
END_VAR
// Ensure there's at least one detail in the step
IF Step.DetailCount < 1 THEN
    IndexConveyorParse := FALSE;
    RETURN;
END_IF

// Use the first detail
Detail := Step.Details[1];

// Check if the detail has enough data fields (we need at least 6 fields)
IF Detail.DataCount < 1 THEN
    IndexConveyorParse := FALSE;
    RETURN;
END_IF

// BoardID
StepOut.ConvIndex := STRING_TO_INT(Detail.Datas[1]);

IndexConveyorParse := TRUE;
END_METHOD

METHOD NailPlateParse : BOOL
VAR_INPUT
    Step    : ST_CSV_Step;
    StepOut : REFERENCE TO ST_Plates;
END_VAR

VAR
    DetailIndex     : INT;
    conversionError : BOOL;
    Detail          : ST_CSV_Detail;
    PlateIndex      : INT;
    TempWidth       : REAL;
    TempHeight      : REAL;
END_VAR
// Ensure there's at least one detail in the step

IF Step.DetailCount < 1 THEN
    NailPlateParse := FALSE;
    RETURN;
END_IF

FOR i := 1 TO Step.DetailCount DO
    Detail := Step.Details[i];

    // Ensure the detail has enough data fields

    IF Detail.DataCount < 11 THEN
        conversionError := TRUE;
        EXIT; // Exit the loop on error
    END_IF;

    // BoardID

    StepOut.Plates[i].BoardID := Detail.Datas[1];

    // PlateID

    StepOut.Plates[i].PlateID := Detail.Datas[2];

    // PlateNumber

    StepOut.Plates[i].PlateNumber := STRING_TO_INT(Detail.Datas[3]);

    // PlateDimensions

    StepOut.Plates[i].PlateDimensions := Detail.Datas[4];

    // PlateGauge

    StepOut.Plates[i].PlateGauge := Detail.Datas[5];

    TempWidth  := STRING_TO_REAL(Detail.Datas[6]);
    TempHeight := STRING_TO_REAL(Detail.Datas[7]);
    // PlateWidth

    StepOut.Plates[i].PlateWidth := MIN(TempWidth, TempHeight);

    // PlateHeight

    StepOut.Plates[i].PlateHeight := MAX(TempWidth, TempHeight);

    // PlatePlaceX

    StepOut.Plates[i].PlatePlaceX := STRING_TO_REAL(Detail.Datas[8]);

    // PlatePlaceY

    StepOut.Plates[i].PlatePlaceY := STRING_TO_REAL(Detail.Datas[9]);

    // PlatePlaceAngle

    StepOut.Plates[i].PlatePlaceAngle := STRING_TO_REAL(Detail.Datas[10]);

    IF TempWidth > TempHeight THEN
        //         StepOut.Plates[i].PlatePlaceAngle := StepOut.Plates[i].PlatePlaceAngle + 90;
        Trace('Width and Height for nailplate swapped');
    END_IF

    // If the value is negative, add 360

    IF StepOut.Plates[i].PlatePlaceAngle < 0 THEN
        StepOut.Plates[i].PlatePlaceAngle := StepOut.Plates[i].PlatePlaceAngle + 360;
    END_IF;

    // TopOrBottom

    StepOut.Plates[i].TopOrBottom := Detail.Datas[11];

END_FOR
END_METHOD

METHOD PickPlaceParse : BOOL
VAR_INPUT
    Step    : ST_CSV_Step;
    StepOut : REFERENCE TO ST_PickPlace;
END_VAR

VAR
    DetailIndex     : INT;
    conversionError : BOOL;
    Detail          : ST_CSV_Detail;
    PlateIndex      : INT;
END_VAR
// Ensure there's at least one detail in the step
IF Step.DetailCount < 1 THEN
    PickPlaceParse := FALSE;
    RETURN;
END_IF

// Ensure the detail has enough data fields
IF Step.Details[1].DataCount < 5 OR Step.Details[2].DataCount < 5 THEN
    conversionError := TRUE;
    PickPlaceParse  := FALSE;
    RETURN; // Exit the loop on error
END_IF;

StepOut.ID        := Step.Details[1].Datas[1];
StepOut.Number    := STRING_TO_INT(Step.Details[1].Datas[2]);
StepOut.Length    := STRING_TO_REAL(Step.Details[1].Datas[3]);
StepOut.Width     := STRING_TO_REAL(Step.Details[1].Datas[4]);
StepOut.boardType := Step.Details[1].Datas[5];

StepOut.XPos      := STRING_TO_REAL(Step.Details[2].Datas[1]);
StepOut.YPos      := STRING_TO_REAL(Step.Details[2].Datas[2]);
StepOut.ZPos      := STRING_TO_REAL(Step.Details[2].Datas[3]);
StepOut.ZRot      := STRING_TO_REAL(Step.Details[2].Datas[4]);
StepOut.ConvIndex := STRING_TO_INT(Step.Details[2].Datas[5]);
END_METHOD

METHOD TrussInfoParse : BOOL
VAR_INPUT
    Step    : ST_CSV_Step;
    StepOut : REFERENCE TO ST_TrussInfo;
END_VAR

VAR
    Detail          : ST_CSV_Detail;
    conversionError : BOOL := FALSE;
END_VAR
// Ensure there's at least one detail in the step
IF Step.DetailCount < 1 THEN
    TrussInfoParse := FALSE;
    RETURN;
END_IF

// Use the first detail
Detail := Step.Details[1];

// Check if the detail has enough data fields (adjust the number based on the fields needed)
IF Detail.DataCount < 9 THEN
    TrussInfoParse := FALSE;
    RETURN;
END_IF

// TrussID
StepOut.TrussID := Detail.Datas[1];

// MemberCount
StepOut.MemberCount := STRING_TO_INT(Detail.Datas[2]);

// TrussXOffs
StepOut.TrussXOffs := STRING_TO_REAL(Detail.Datas[3]);

// TrussYOffs
StepOut.TrussYOffs := STRING_TO_REAL(Detail.Datas[4]);

// TrussLength
StepOut.TrussLength := STRING_TO_REAL(Detail.Datas[5]);

// TrussWidth
StepOut.TrussWidth := STRING_TO_REAL(Detail.Datas[6]);

// PressBeforeTruss
// Assuming that the data is "1" = 'TRUE' or "0" = 'FALSE' as strings
IF Detail.Datas[7] = '1' THEN
    StepOut.PressBeforeTruss := TRUE;
ELSE
    StepOut.PressBeforeTruss := FALSE;
END_IF

// LeftEndType
StepOut.LeftEndType := Detail.Datas[8];

// RightEndType
StepOut.RightEndType := Detail.Datas[9];

TrussInfoParse := TRUE;
END_METHOD

//! @summary This method serves as the entry point for all underlying FB logic

//! @description This method should be called cyclically by descendant function blocks by invoking <c>SUPER^.CyclicLogic()</c>.  Alternatively, the contents of this method could be reimplemented entirely in which case a call to this method would not be necessary.
METHOD PUBLIC CyclicLogic
VAR
    i : UDINT;
END_VAR

VAR_INST
    test_header   : STRING          := 'Header';
    test_header2  : STRING          := 'Header';
    test_header3  : STRING          := 'Header';
    test_message1 : STRING          := 'message 1';
    test_message2 : STRING          := 'message 2 ';
    test_message3 : STRING          := 'message 3';
    test_message4 : STRING          := 'message 4';
    test_message5 : STRING          := 'message 5';
    test_message6 : STRING          := 'message 6';
    test_message7 : STRING          := 'message 7';
    test_btn1     : STRING          := 'Btn 1';
    test_btn2     : STRING          := 'Btn 2';
    test_btn3     : STRING          := 'Btn 3';
    test_btn4     : STRING          := 'Btn 4';
    test_btn5     : STRING          := 'Btn 5';
    test_severity : TcEventSeverity := 1;
    test_icon     : USINT           := 1;
    result        : USINT;

    MsgBox_R_TRIG : R_TRIG;
END_VAR
//HMI control for EM

fbControlSourceHMI.CyclicLogic();
MessageBox_Data.ErrorPresent := FALSE;

SUPER^.CyclicLogic();
MessageBox_Data.Equipment_Module        := _EquipmentModuleID;
MessageBox_Data.Equipment_Module_String := THIS^._Name;
test_header                             := CONCAT(THIS^._Name, ' -> header');
test_header                             := CONCAT(test_header, ' MsgBox1');
test_header2                            := CONCAT(test_header, ' MsgBox2');
// test_header3                            := CONCAT(test_header, ' MsgBox3');

MsgBox_R_TRIG(CLK := Global.testmessagebox);

IF MsgBox_R_TRIG.Q THEN
    testmessagebox2 := TRUE;
END_IF

IF testmessagebox2 OR MsgBox_R_TRIG.Q THEN
    result := RaiseMessageBox(Header   := test_header2,
                              Message1 := test_message1,
                              Message2 := test_message2,
                              Message3 := test_message3,
                              Message4 := test_message4,
                              Message5 := test_message5,
                              Message6 := test_message6,
                              Message7 := test_message7,
                              Btn1     := test_btn1,
                              Btn2     := test_btn2,
                              Btn3     := test_btn3,
                              Btn4     := test_btn4,
                              Btn5     := test_btn5,
                              Severity := test_severity,
                              Icon     := test_icon);

    IF result > 0 THEN
        testmessagebox2 := FALSE;
    END_IF
END_IF

IF _CurrentState = E_PMLState.ePMLState_Suspended THEN
    AutoUnsuspendCheck_TON(IN := TRUE, PT := T#500MS);
    AutoUnsuspendReset_TON(IN := FALSE, PT := T#5S);
ELSIF _CurrentState = E_PMLState.ePMLState_Execute THEN
    AutoUnsuspendCheck_TON(IN := FALSE, PT := T#500MS);
    AutoUnsuspendReset_TON(IN := TRUE, PT := T#5S);

    IF AutoUnsuspendReset_TON.Q THEN
        AutoUnsuspendAvailable := TRUE;
    END_IF
END_IF

IF _CurrentState = E_PMLState.ePMLState_Held OR
   _CurrentState = E_PMLState.ePMLState_Suspended OR
   _CurrentState = E_PMLState.ePMLState_Idle OR
   _CurrentState = E_PMLState.ePMLState_stopped OR
   _CurrentState = E_PMLState.ePMLState_Aborted THEN
    HMIControl();
END_IF

IF testbool5 THEN
    teststring := LengthFormatString(testlreal);
    testbool5  := FALSE;
END_IF

SubModuleMonitor();
ComponentMonitor();
EM_BufferLogging(sNetID := '', nDBID := 2, bRecord := testbool9);
END_METHOD

METHOD CyclicLogicSimulation : BOOL
VAR_INPUT
END_VAR
// AllowHMIControl(ThisModuleOnly:=FALSE); //Allow control for recovery
END_METHOD

PROPERTY Step : DINT
SET
_Step := Step;
END_SET
END_PROPERTY

METHOD AssignMessageBox
VAR_INPUT
    MsgBox_Data     : REFERENCE TO ST_MessageBox_Data;
    MsgBox_Response : REFERENCE TO ST_MessageBox_Response;
END_VAR
MsgBox_Data         := MessageBox_Data;
MessageBox_Response := MsgBox_Response;
END_METHOD

//! @summary This method monitors <b>components</b> within this PackML module and initiates fault responses as required
METHOD PROTECTED ComponentMonitor : BOOL
VAR
    AlarmResponses : ARRAY[0..4] OF E_AlarmResponse; //Temporary response array
    i              : UDINT;
END_VAR

//! @description This method is called cyclically by <c>CyclicLogic()</c>
FOR i := 1 TO NumberOfComponents DO
    IF _CurrentState <> E_PMLState.ePMLState_Aborted AND
       _CurrentState <> E_PMLState.ePMLState_Aborting AND
       _CurrentState <> E_PMLState.ePMLState_Clearing AND
       _CurrentState <> E_PMLState.ePMLState_Suspended AND
       _CurrentState <> E_PMLState.ePMLState_Unsuspending AND
       _CurrentState <> E_PMLState.ePMLState_Held AND
       _CurrentState <> E_PMLState.ePMLState_Unholding AND
       _CurrentState <> E_PMLState.ePMLState_Stopped AND
       _CurrentState <> E_PMLState.ePMLState_Stopping THEN
        AlarmResponses := ipComponents[i].ParentResponseDefinitions;

        CASE AlarmResponses[ipComponents[i].CurrentAlarmSeverity] OF
            E_AlarmResponse.Abort_ImmediateError:
                SuspendImmediate();

            E_AlarmResponse.Abort_Immediate:
                SuspendControlled();

            E_AlarmResponse.Stop_Immediate:
                StopImmediate();

            E_AlarmResponse.Stop_Controlled:
                StopControlled();

            E_AlarmResponse.Hold_Immediate:
                HoldImmediate();

            E_AlarmResponse.Hold_Controlled:
                HoldControlled();

            E_AlarmResponse.Suspend_Immediate:
                SuspendImmediate();

            E_AlarmResponse.Suspend_Controlled:
                SuspendControlled();

            E_AlarmResponse.NoResponse:
                ;
        END_CASE
    ELSIF _CurrentState = E_PMLState.ePMLState_Stopped OR _CurrentState = E_PMLState.ePMLState_Stopping THEN
        AlarmResponses := ipComponents[i].ParentResponseDefinitions;

        CASE AlarmResponses[ipComponents[i].CurrentAlarmSeverity] OF
            E_AlarmResponse.Abort_ImmediateError:
                AbortImmediateError(ipComponents[i].Name, FALSE);

            E_AlarmResponse.Abort_Immediate:
                AbortImmediate();

            E_AlarmResponse.NoResponse:
                ;
        END_CASE
    END_IF
END_FOR
END_METHOD

METHOD EM_BufferLogging
VAR_INPUT
    sNetID  : T_AmsNetID;
    nDBID   : UDINT;
    bRecord : BOOL;
END_VAR

VAR_OUTPUT
    bTableCreated : BOOL;
    bRecording    : BOOL;
    bError        : BOOL;
    sTableName    : T_MaxString;
    nRecords      : ULINT;
END_VAR
//Create timestamp
fbGetSystemTime1(timeLoDW => dwTimeLoDW, timeHiDW => dwTimeHiDW);
tFileTime.dwLowDateTime  := dwTimeLoDW;
tFileTime.dwHighDateTime := dwTimeHiDW;
MEMCPY(ADR(nTimestamp), ADR(tFileTime), 8);

CASE nState OF
    0: //Init

        IF bRecord THEN
            bError        := FALSE;
            bTableCreated := FALSE;
            bRecording    := FALSE;
            nRecords      := 0;

            sTableName := 'em_log';

            sCmd1 := CONCAT('INSERT INTO ', sTableName);
			
            sCmd2 := ' (timestamp,module,state,msg) VALUES({Timestamp},{ModuleName},{PackMLState},{Message});';

            CONCAT2(ADR(sCmd1), ADR(sCmd2), ADR(sCmd), SIZEOF(sCmd));

            nWriteBufferIndex := 0;
            nWriteIndex       := 0;
            nSQLIndex         := 0;

            nState := 2;
        END_IF

    2: //Recording		
        bRecording := TRUE;

        fbGetSystemTime(timeLoDW => fileTime.dwLowDateTime, timeHiDW => fileTime.dwHighDateTime);
        dtTime := FILETIME_TO_DT(fileTime);

		aPara[0].eParaType := E_ExpParameterType.DateTime;
		aPara[0].nParaSize := 4;
		aPara[0].sParaName := 'timestamp';

		aPara[1].eParaType := E_ExpParameterType.STRING_;
		aPara[1].nParaSize := 33;
		aPara[1].sParaName := 'module';

		aPara[2].eParaType := E_ExpParameterType.STRING_;
		aPara[2].nParaSize := 33;
		aPara[2].sParaName := 'state';

		aPara[3].eParaType := E_ExpParameterType.STRING_;
		aPara[3].nParaSize := 256;
		aPara[3].sParaName := 'msg';

        //Fill buffer
        stData[nWriteBufferIndex, nWriteIndex].Timestamp   := dtTime;
        stData[nWriteBufferIndex, nWriteIndex].ModuleName  := THIS^.Name;
        stData[nWriteBufferIndex, nWriteIndex].PackMLState := TO_STRING(_CurrentState);
        stData[nWriteBufferIndex, nWriteIndex].Message     := CONCAT(INT_TO_STRING(nWriteBufferIndex), CONCAT(':  ', INT_TO_STRING(nWriteIndex)));

        //Set buffer index
        nWriteIndex := nWriteIndex + 1;

        IF nWriteIndex = 100 THEN
            nWriteIndex                  := 0;
            aWriteSQL[nWriteBufferIndex] := TRUE;
            nWriteBufferIndex            := nWriteBufferIndex + 1;

            IF nWriteBufferIndex = 20 THEN
                nWriteBufferIndex := 0;
            END_IF

            IF aWriteSQL[nWriteBufferIndex] THEN
                nState := 255;
                RETURN;
            END_IF
        END_IF

        //Write buffer element (100 samples) to database
        IF aWriteSQL[nSQLIndex] THEN
            IF fbPLCDBCmd.Execute(nDBID,
                                  ADR(sCmd),
                                  SIZEOF(sCmd),
                                  ADR(stData[nSQLIndex, 0]),
                                  SIZEOF(stData[nSQLIndex, 0]) * 100,
                                  ADR(aPara),
                                  SIZEOF(aPara)) THEN
                IF fbPLCDBCmd.bError THEN
					tcMessage := fbPLCDBCmd.ipTcResult;
                    nState := 255;
                ELSE
                    nRecords := nRecords + 100;

                    aWriteSQL[nSQLIndex] := FALSE;

                    nSQLIndex := nSQLIndex + 1;

                    IF nSQLIndex = 20 THEN
                        nSQLIndex := 0;
                    END_IF

                    IF NOT bRecord THEN
                        bRecording := FALSE;
                        nState     := 0;
                    END_IF
                END_IF
            END_IF
        END_IF

    255: //Error
        bError     := TRUE;
        bRecording := FALSE;

        IF NOT bRecord THEN
            nState := 0;
        END_IF
END_CASE
END_METHOD

METHOD HMIControl
VAR_INPUT
END_VAR
END_METHOD

(*
	This method takes an input of LREAL length in mm and converts it to a string of the board print format of FT:IN:16th
*)
METHOD LengthFormatString : STRING
VAR_INPUT
    BoardLength : LREAL;
END_VAR

VAR
    temp_lreal  : LREAL;
    temp_in     : LREAL;
    temp_in_dec : LREAL;
    temp_ft     : LREAL;
    temp_16     : LREAL;
    tempstring  : STRING;
    ft          : LREAL;
    in          : LREAL;
    sixteenth   : LREAL;
END_VAR
temp_ft     := BoardLength / 25.4 / 12;
ft          := TRUNC(temp_ft);
temp_in_dec := temp_ft - ft;
temp_in     := temp_in_dec * 12;
in          := TRUNC(temp_in);
temp_16     := temp_in - in;
sixteenth   := TRUNC((temp_16 * 16) + 0.5);

IF sixteenth = 16 THEN
    in        := in + 1;
    sixteenth := 0;
END_IF

IF in = 12 THEN
    ft := ft + 1;
    in := 0;
END_IF

LengthFormatString := concat(USINT_TO_STRING(LREAL_TO_USINT(ft)),
                             Concat(':', CONCAT(USINT_TO_STRING(LREAL_TO_USINT(in)), CONCAT(':', USINT_TO_STRING(LREAL_TO_USINT(sixteenth))))));
END_METHOD

METHOD MotorResetAndEnable : BOOL
VAR_INPUT
    Motor : REFERENCE TO FB_Component_BasicSlaveAxis;
END_VAR
MotorResetAndEnable := FALSE;

IF Motor.Error THEN
    Motor.Reset();
ELSE

    Motor.Enable();

    IF Motor.Enabled THEN
        MotorResetAndEnable := TRUE;
    END_IF
END_IF
END_METHOD

METHOD MotorsHome : BOOL
VAR_INPUT
END_VAR
MotorsHome := TRUE;
END_METHOD

METHOD MotorsInit : BOOL
VAR_INPUT
END_VAR
MotorsInit := TRUE;
END_METHOD

METHOD MotorsInitAlignGearIn : BOOL
VAR_INPUT
END_VAR
MotorsInitAlignGearIn := TRUE;
END_METHOD

METHOD RaiseAlarm2Args
VAR_IN_OUT
    fbAlarm : FB_TcAlarm; //Alarm to be raised
END_VAR

VAR_INPUT
    String_1 : STRING; //First String Parameter (The Name of this component will be applied first automatically)
    String_2 : STRING; //Second String Parameter
END_VAR
F_RaiseAlarmWithStringParameters(Alarm := fbAlarm, String_1 := Name, String_2 := String_1, String_3 := String_2);
END_METHOD

METHOD RaiseMessageBox : USINT
VAR_INPUT
    Header   : STRING;
    Message1 : STRING;
    Message2 : STRING          := '';
    Message3 : STRING          := '';
    Message4 : STRING          := '';
    Message5 : STRING          := '';
    Message6 : STRING          := '';
    Message7 : STRING          := '';
    Btn1     : STRING          := '';
    Btn2     : STRING          := '';
    Btn3     : STRING          := '';
    Btn4     : STRING          := '';
    Btn5     : STRING          := '';
    Severity : TcEventSeverity := TcEventSeverity.Info;
    Icon     : USINT           := 1;
END_VAR

VAR_INST
    TimeStampTrig : R_TRIG;
    MsgBox_Raised : BOOL;
END_VAR

VAR
    fbGetSystemTime : GETSYSTEMTIME;
    fileTime        : T_FILETIME;
    tempDT          : DT;
    tempTOD         : TOD;
    tempTODString   : STRING;
    sTime           : STRING;
    ResponseString  : STRING;
END_VAR
RaiseMessageBox := 0;
fbGetSystemTime(timeLoDW => fileTime.dwLowDateTime, timeHiDW => fileTime.dwHighDateTime);

IF MessageBox_Response.ErrorAcknowledge = TRUE AND MessageBox_Response.ErrorSolution > 0 AND MessageBox_Data.Header = Header THEN
    RaiseMessageBox := MessageBox_Response.ErrorSolution;

    CASE RaiseMessageBox OF
        1:
            ResponseString := Btn1;

        2:
            ResponseString := Btn2;

        3:
            ResponseString := Btn3;

        4:
            ResponseString := Btn4;

        5:
            ResponseString := Btn5;
    END_CASE

    Trace(CONCAT('Msg Cleared: ', CONCAT(Header, CONCAT('; Response: ', ResponseString))));
    ResetMessageBox();
    TimeStampTrig(CLK := FALSE);
ELSE
    IF Header <> '' AND
       Message1 <> '' AND
       (Btn1 <> '' OR Btn2 <> '' OR Btn3 <> '' OR Btn4 <> '' OR Btn5 <> '') AND
       (MessageBox_Response.ErrorRaised = FALSE OR MessageBox_Data.Header = Header) THEN
        TimeStampTrig(CLK := TRUE);
        MessageBox_Data.Header := Header;

        IF TimeStampTrig.Q THEN
            tempDT                    := SYSTEMTIME_TO_DT(FILETIME_TO_SYSTEMTIME(fileTime));
            tempTOD                   := DT_TO_TOD(tempDT);
            tempTODString             := TOD_TO_STRING(tempTOD);
            MessageBox_Data.TimeStamp := REPLACE(tempTODString, '', 1, 4);
            Trace(CONCAT('Msg Raised: ', Header));
        END_IF

        MessageBox_Data.Icon := Icon;

        MessageBox_Data.Messages.Message1 := Message1;
        MessageBox_Data.Messages.Message2 := Message2;
        MessageBox_Data.Messages.Message3 := Message3;
        MessageBox_Data.Messages.Message4 := Message4;
        MessageBox_Data.Messages.Message5 := Message5;
        MessageBox_Data.Messages.Message6 := Message6;
        MessageBox_Data.Messages.Message7 := Message7;

        MessageBox_Data.Buttons.Button1.Text := Btn1;
        MessageBox_Data.Buttons.Button2.Text := Btn2;
        MessageBox_Data.Buttons.Button3.Text := Btn3;
        MessageBox_Data.Buttons.Button4.Text := Btn4;
        MessageBox_Data.Buttons.Button5.Text := Btn5;

        IF MessageBox_Data.Buttons.Button1.Text <> '' THEN
            MessageBox_Data.Buttons.Button1.Visible := TRUE;
        ELSE
            MessageBox_Data.Buttons.Button1.Visible := FALSE;
        END_IF

        IF MessageBox_Data.Buttons.Button2.Text <> '' THEN
            MessageBox_Data.Buttons.Button2.Visible := TRUE;
        ELSE
            MessageBox_Data.Buttons.Button2.Visible := FALSE;
        END_IF

        IF MessageBox_Data.Buttons.Button3.Text <> '' THEN
            MessageBox_Data.Buttons.Button3.Visible := TRUE;
        ELSE
            MessageBox_Data.Buttons.Button3.Visible := FALSE;
        END_IF

        IF MessageBox_Data.Buttons.Button4.Text <> '' THEN
            MessageBox_Data.Buttons.Button4.Visible := TRUE;
        ELSE
            MessageBox_Data.Buttons.Button4.Visible := FALSE;
        END_IF

        IF MessageBox_Data.Buttons.Button5.Text <> '' THEN
            MessageBox_Data.Buttons.Button5.Visible := TRUE;
        ELSE
            MessageBox_Data.Buttons.Button5.Visible := FALSE;
        END_IF

        MessageBox_Data.Severity := Severity;

        MessageBox_Data.ErrorPresent := TRUE;
    ELSE
        //can't raise message with no header, message, or at least one button to clear message. 
    END_IF

END_IF
END_METHOD

METHOD PROTECTED RegisterSubmodules
VAR_INPUT
    SubModule : I_EquipmentModule_SR;
END_VAR

VAR
    i       : UDINT;
    PLCStop : PLC_Stop;
END_VAR
IF NOT _InitComplete AND (SubModule <> 0) THEN
    FOR i := 1 TO SPT_BaseTypes.Parameters_PackML_Base.MAX_NO_OF_SUBMODULES DO
        IF ipSubModules_SR[i] = SubModule THEN
            //Submodule already registered
            RETURN;
        END_IF
    END_FOR

    FOR i := 1 TO SPT_BaseTypes.Parameters_PackML_Base.MAX_NO_OF_SUBMODULES DO
        IF ipSubModules_SR[i] = 0 THEN
            ipSubModules_SR[i] := SubModule;
            ipSubModules[i]    := SubModule;
            RETURN;
        END_IF
    END_FOR

    //If we get here then we are exceeding the array bounds
    Trace(CONCAT('***CRITICAL - Failed to register SubModule!!  (', CONCAT(SubModule.Name, ')***')));
    PLCStop(STOP := TRUE);

END_IF
END_METHOD

METHOD ResetMessageBox
VAR_INPUT
END_VAR

VAR
    EmptyMessageBox : ST_MessageBox_Data;
END_VAR
MessageBox_Data := EmptyMessageBox;
END_METHOD

METHOD ResetOnResume : BOOL
VAR_INPUT
END_VAR
IF ResetComponents() THEN
    _ComponentsReset := TRUE;
END_IF

IF _ComponentsReset THEN
    ClearAlarms(EquipmentModule_Alarms);
    ResetOnResume := TRUE;
END_IF
END_METHOD

METHOD RestartStateCheck
VAR_INPUT
END_VAR
END_METHOD

METHOD SimHoming : BOOL
VAR_INPUT
    Motor  : REFERENCE TO FB_Component_BasicSlaveAxis_SoE;
    SimPos : LREAL;
END_VAR

VAR_INST
    _SimHomingState : USINT;
    _SetPositionSim : FB_HomeRoutine_SetPosition;
END_VAR
CASE _SimHomingState OF
    0:
        SimHoming                    := FALSE;
        Motor.HomeMethod             := _SetPositionSim;
        _SetPositionSim.HomePosition := SimPos;
        _SetPositionSim.Execute();
        _SimHomingState := 10;

    10:
        IF _SetPositionSim.Busy = FALSE AND ABS(Motor.ActualPosition - SimPos) < 0.0001 THEN
            _SimHomingState := 20;
        END_IF

    20:
        SimHoming       := TRUE;
        _SimHomingState := 0;
END_CASE
END_METHOD

//! @summary This method monitors <b>submodules</b> within this PackML module and initiates fault responses as required
METHOD PROTECTED SubModuleMonitor : BOOL
VAR
    AlarmResponses : ARRAY[0..4] OF E_AlarmResponse; //Temporary response array	
    i              : UDINT;
END_VAR

//! @description This method is called cyclically by <c>CyclicLogic()</c>
FOR i := 1 TO NumberOfSubModules DO
    IF _CurrentState <> E_PMLState.ePMLState_Aborted AND
       _CurrentState <> E_PMLState.ePMLState_Aborting AND
       _CurrentState <> E_PMLState.ePMLState_Clearing AND
       _CurrentState <> E_PMLState.ePMLState_Stopped AND
       _CurrentState <> E_PMLState.ePMLState_Stopping THEN
        AlarmResponses := ipSubModules[i].ParentResponseDefinitions;

        CASE AlarmResponses[ipSubModules[i].CurrentAlarmSeverity] OF
            E_AlarmResponse.Abort_ImmediateError:
                SuspendImmediate();

            E_AlarmResponse.Abort_Immediate:
                SuspendControlled();

            E_AlarmResponse.Stop_Immediate:
                StopImmediate();

            E_AlarmResponse.Stop_Controlled:
                StopControlled();

            E_AlarmResponse.Hold_Immediate:
                HoldImmediate();

            E_AlarmResponse.Hold_Controlled:
                HoldControlled();

            E_AlarmResponse.Suspend_Immediate:
                SuspendImmediate();

            E_AlarmResponse.Suspend_Controlled:
                SuspendControlled();

            E_AlarmResponse.NoResponse:
                ;
        END_CASE
    ELSIF _CurrentState = E_PMLState.ePMLState_Stopped OR _CurrentState = E_PMLState.ePMLState_Stopping THEN
        AlarmResponses := ipSubModules[i].ParentResponseDefinitions;

        CASE AlarmResponses[ipSubModules[i].CurrentAlarmSeverity] OF
            E_AlarmResponse.Abort_ImmediateError:
                AbortImmediateError(ipSubModules[i].Name, TRUE);

            E_AlarmResponse.Abort_Immediate:
                AbortImmediate();

            E_AlarmResponse.NoResponse:
                ;
        END_CASE
    END_IF
END_FOR
END_METHOD

METHOD TorqueHoming : BOOL
VAR_INPUT
    Motor      : REFERENCE TO FB_Component_BasicSlaveAxis_SoE;
    HomingInfo : REFERENCE TO ST_HomingParams;
    Velocity   : LREAL;
    Torque     : LREAL;
    Direction  : SPT_Motion_Control.MC_Home_Direction;
END_VAR

VAR
    McReadParam_Bias    : INT;
    CurrentPositionBias : INT;
    ParameterNumber     : INT;
    Axis                : INT;
    Value               : INT;
END_VAR
TorqueHoming := FALSE;

CASE HomingInfo.HomingState OF
    0:
        HomingInfo.TorqueControl(Axis              := Motor.Axis,
                                 Execute           := FALSE,
                                 Relative          :=,
                                 Torque            := Torque,
                                 TorqueRamp        := 50,
                                 VelocityLimitHigh := Velocity,
                                 VelocityLimitLow  := -Velocity,
                                 BufferMode        :=,
                                 Options           := HomingInfo.TorqueControlParams);

        HomingInfo.Execute_WriteLimit := FALSE;

        HomingInfo.TorqueControlParams.EnableManualTorqueStartValue := TRUE;
        HomingInfo.TorqueControlParams.ManualTorqueStartValue       := Motor.Axis.NcToPlc.ActTorque;

        IF Direction = SPT_Motion_Control.MC_Home_Direction.mcPositiveDirection THEN
            HomingInfo.SetPositionHomingRoutine.HomePosition := HomingInfo.HomePosMax;
        ELSE
            HomingInfo.SetPositionHomingRoutine.HomePosition := HomingInfo.HomePosMin;
        END_IF

        Motor.HomeMethod       := HomingInfo.SetPositionHomingRoutine;
        HomingInfo.HomingState := 1;

    1:
        // Ensure Motors are enabled before homing

        IF Motor.Error THEN
            Motor.Reset();
        ELSE
            HomingInfo.HomingState := 2;
        END_IF

    2:
        Motor.GearOut();

        IF Motor.InGear = FALSE THEN
            HomingInfo.HomingState := 3;
        END_IF

    3:
        // Ensure Motors are enabled before homing

        Motor.Enable();

        IF Motor.Enabled THEN
            HomingInfo.HomingState := 5;
        END_IF

    5:
        HomingInfo.Execute_WriteLimit := TRUE;
        HomingInfo.EnablePosLim       := FALSE;
        HomingInfo.EnableNegLim       := FALSE;

        IF HomingInfo.WritePosLim.Done AND HomingInfo.WriteNegLim.Done THEN
            HomingInfo.HomingState        := 10;
            HomingInfo.Execute_WriteLimit := FALSE;

        END_IF

    10:
        // Execute hard stop home for top and bottom carriages

        HomingInfo.TorqueControl(Axis              := Motor.Axis,
                                 Execute           := TRUE,
                                 Relative          :=,
                                 Torque            := Torque,
                                 TorqueRamp        := 50,
                                 VelocityLimitHigh := Velocity,
                                 VelocityLimitLow  := -Velocity,
                                 BufferMode        :=,
                                 Options           := HomingInfo.TorqueControlParams);

        HomingInfo.HomingTON(IN := ABS(Motor.Axis.NcToPlc.ActTorque - Torque) < 0.5 AND (Motor.ActualVelocity < 0.2), PT := T#100MS);

        IF HomingInfo.HomingTON.Q THEN
            HomingInfo.HomingState := 20;
        END_IF

    20:
        IF Motor.Stop() THEN
            HomingInfo.HomingState := 30;
        END_IF

    30:
        IF Motor.Home() THEN
            HomingInfo.HomingState := 40;
        END_IF

    40:
        // Wait for hard stop homing routines to complete

        Motor.Axis.ReadStatus();

        IF (Motor.Axis.NcToPlc.ActPos - HomingInfo.SetPositionHomingRoutine.HomePosition) < 1 THEN
            IF NOT Motor.Error THEN
                HomingInfo.HomingState := 50;
            ELSE
                HomingInfo.HomingState := 5000;
            END_IF
        END_IF

    50:
        //         Motor.Disable();
        // 
        //         IF Motor.Enabled = FALSE THEN
        //             HomingInfo.HomingState := 60;
        //         END_IF
        // 
        //     60:
        //         HomingInfo.SetPositionOffset(Axis     := Motor.Axis,
        //                                      Execute  := TRUE,
        //                                      Position := Motor.Axis.NcToPlc.ActPos,
        //                                      Relative := FALSE,
        //                                      Feedback := SPT_Motion_Control.E_PositionOffsetFeedback.ePositionOffsetFeedback1,
        //                                      Memory   := SPT_Motion_Control.E_PositionOffsetMemory.ePositionOffsetMemory_Drive);
        // 
        //         IF HomingInfo.SetPositionOffset.Busy = FALSE THEN
        //             HomingInfo.HomingState := 70;
        //         END_IF
        // 
        //     70:
        // Re-enable the Motors
        HomingInfo.Execute_WriteLimit := TRUE;
        HomingInfo.EnablePosLim       := TRUE;
        HomingInfo.EnableNegLim       := TRUE;

        IF HomingInfo.WritePosLim.Done AND HomingInfo.WriteNegLim.Done THEN
            HomingInfo.HomingState        := 80;
            HomingInfo.Execute_WriteLimit := FALSE;

        END_IF

    80:
        Motor.Enable();

        IF Motor.Enabled THEN
            HomingInfo.HomingState := 90;
        END_IF

    90:
        // Move to set position after homing

        TorqueHoming           := TRUE;
        HomingInfo.HomingState := 0;

    5000:
        Motor.Stop();

    // Error in homing routine

    {warning:error in homing routine}
END_CASE

HomingInfo.WritePosLim(Axis            := Motor.Axis,
                       Execute         := HomingInfo.Execute_WriteLimit,
                       ParameterNumber := SPT_Motion_Control.MC_AxisParameter.EnableLimitPos,
                       Value           := HomingInfo.EnablePosLim);

HomingInfo.WriteNegLim(Axis            := Motor.Axis,
                       Execute         := HomingInfo.Execute_WriteLimit,
                       ParameterNumber := SPT_Motion_Control.MC_AxisParameter.EnableLimitNeg,
                       Value           := HomingInfo.EnableNegLim);
END_METHOD

METHOD TorqueHoming_old : BOOL
VAR_INPUT
    Motor      : REFERENCE TO FB_Component_BasicSlaveAxis_SoE;
    HomingInfo : REFERENCE TO ST_HomingParams;
    lag        : LREAL;
    velocity   : LREAL;
    torque     : LREAL;
    Direction  : SPT_Motion_Control.MC_Home_Direction;
END_VAR

VAR
    McReadParam_Bias    : INT;
    CurrentPositionBias : INT;
    ParameterNumber     : INT;
    Axis                : INT;
    Value               : INT;
END_VAR
CASE HomingInfo.HomingState OF
    0:
        Motor.HomeMethod := HomingInfo.HardStopHomingRoutine;

        // Init homing parameters for Hard Stop

        //         HomingInfo.HardStopHomingParams.DisableDriveAccess     := TRUE;
        HomingInfo.HardStopHomingParams.Acceleration           := velocity * 2;
        HomingInfo.HardStopHomingParams.Deceleration           := velocity * 2;
        HomingInfo.HardStopHomingParams.Direction              := Direction;
        HomingInfo.HardStopHomingParams.DistanceLimit          := 10000;
        HomingInfo.HardStopHomingParams.LagLimit               := lag;
        HomingInfo.HardStopHomingParams.TorqueLimit            := torque;
        HomingInfo.HardStopHomingParams.TimeLimit              := TIME#60S0MS;
        HomingInfo.HardStopHomingParams.Velocity               := velocity;
        HomingInfo.HardStopHomingParams.DetectionVelocityLimit := velocity * 1.5;
        HomingInfo.HardStopHomingParams.DetectionVelocityTime  := T#400MS;
        HomingInfo.HardStopHomingRoutine.CyclicLogic();

        IF Direction = SPT_Motion_Control.MC_Home_Direction.mcPositiveDirection THEN
            HomingInfo.HardStopHomingRoutine.HomePosition := HomingInfo.HomePosMax;
        ELSE
            HomingInfo.HardStopHomingRoutine.HomePosition := HomingInfo.HomePosMin;
        END_IF

        HomingInfo.HardStopHomingRoutine.Parameters := HomingInfo.HardStopHomingParams;
        HomingInfo.HomingState                      := 1;

    1:
        // Ensure Motors are enabled before homing

        IF Motor.Error THEN
            Motor.Reset();
        ELSE
            HomingInfo.HomingState := 2;
        END_IF

    2:
        Motor.GearOut();

        IF Motor.InGear = FALSE THEN
            HomingInfo.HomingState := 3;
        END_IF

    3:
        // Ensure Motors are enabled before homing

        Motor.Enable();

        IF Motor.Enabled THEN
            HomingInfo.HomingState := 10;
        END_IF

    10:
        // Execute hard stop home for top and bottom carriages

        IF Motor.Home() THEN
            HomingInfo.HomingState := 20;
        END_IF

    20:
        // Wait for hard stop homing routines to complete

        IF Motor.Axis.Status.Homed THEN
            IF NOT Motor.Error THEN
                HomingInfo.HomingState := 21;
            ELSE
                HomingInfo.HomingState := 5000;
            END_IF
        END_IF

    21:
        //         Motor.Disable();

        // 

        //         IF Motor.Enabled = FALSE THEN

        //             HomingInfo.HomingState := 22;

        //         END_IF

        // 

        //     22:

        // 

        HomingInfo.SetPositionOffset(Axis     := Motor.Axis,
                                     Execute  := TRUE,
                                     Position := HomingInfo.HardStopHomingRoutine.HomePosition,
                                     Relative := FALSE,
                                     Feedback := SPT_Motion_Control.E_PositionOffsetFeedback.ePositionOffsetFeedback1,
                                     Memory   := SPT_Motion_Control.E_PositionOffsetMemory.ePositionOffsetMemory_Drive);

        IF HomingInfo.SetPositionOffset.Busy = FALSE THEN
            HomingInfo.HomingState := 23;
        END_IF

    23:
        //         Motor.HomeMethod := HomingInfo.AbsHomingRoutine;

        //         HomingInfo.AbsHomingRoutine.Parameters REF= HomingInfo.AbsHomingParams;

        //         HomingInfo.AbsHomingRoutine.Execute();

        // 

        //         HomingInfo.ReadParams(ParameterNumber:=MC_AxisParameter.AxisEncoderOffset,

        //                               Axis           :=Motor.Axis,

        //                               Value          =>HomingInfo.HomingBias);

        // 

        HomingInfo.HomingState := 30;

    30:
        // Re-enable the Motors

        Motor.Enable();

        IF Motor.Enabled THEN
            HomingInfo.HomingState := 40;
        END_IF

    40:
        // Move to set position after homing

        TorqueHoming_old       := TRUE;
        HomingInfo.HomingState := 0;

    5000:
        Motor.Stop();

    // Error in homing routine

    {warning:error in homing routine}
END_CASE
END_METHOD

METHOD WaitSync_Handler : BOOL
VAR_INPUT
    WaitSync : E_WaitSync;
END_VAR

VAR_OUTPUT
    WaitSyncResponse : E_WaitSync;
END_VAR

VAR_INST
    State : UDINT;
END_VAR
WaitSync_Handler := FALSE;
WaitSyncResponse := _ResponseWaitSync;

CASE State OF
    0:
        IF WaitSync > E_WaitSync.EMPTY THEN
            State := 1;
        END_IF

    1:
        _RequestedWaitSync := WaitSync;

        IF _RequestedWaitSync = _ResponseWaitSync THEN
            State := 2;
        END_IF

    2:
        _RequestedWaitSync := E_WaitSync.EMPTY;

        IF _ResponseWaitSync = E_WaitSync.EMPTY THEN
            WaitSync_Handler := TRUE;
            State            := 0;
        END_IF

END_CASE
END_METHOD

METHOD WaitSync_ReadWrite : BOOL
VAR_INPUT
    request  : REFERENCE TO E_WaitSync;
    response : REFERENCE TO E_WaitSync;
END_VAR
WaitSync_ReadWrite := FALSE;

request           := _RequestedWaitSync;
_ResponseWaitSync := response;
END_METHOD

METHOD WaitSyncCheck : BOOL
VAR_INPUT
    Request : E_WaitSync;
END_VAR
WaitSyncCheck := FALSE;

_RequestedWaitSync := Request;

IF _ResponseWaitSync = Request THEN
    WaitSyncCheck := TRUE;
END_IF
END_METHOD

//! @summary This method contains code which will execute when this PackML module is in the <b>Holding</b> state
METHOD PROTECTED Holding
VAR
    i               : UDINT;
    SubModulesReady : BOOL := TRUE;
END_VAR

(*! <description><b>Note:</b> The <i>Hold</i> command is intended to be given by an operator. It is meant to be distinct from a <i>Suspend</i> in that upstream/downstream jams, etc. should be handled automatically using <i>Suspend</i>.  Both <i>Hold</i>and<i>Suspend</i> result in a <i>paused</i> state which should allow resumption of the <b>Execute</b> state. 
<table> 
	<tr>
		<th> Previous State </th>
		<th> Transition In </th>
		<th> Transition Out </th>
		<th> Next State  </th> 
	</tr>
	<tr>
		<td> Execute </td>
		<td> Hold Command </td> 
		<td> State Complete </td>
		<td> Held </td> 
	</tr>
</table>
This method is called as required by <c>StateControl()</c>
</description> 

*)
_MotorsReset      := FALSE;
_MotorInitState   := 0;
_ComponentsReset  := FALSE;
_AlignGearInState := 0;
_Handshake_State  := 0;

SUPER^.Holding();
END_METHOD

//! @summary This method contains code which will execute when this PackML module is in the <b>Resetting</b> state
METHOD PROTECTED Resetting
VAR
    i               : UDINT;
    SubModulesReady : BOOL := TRUE;
END_VAR

(*! <description> <b>Note:</b> The <i>Reset</i> command can also be thought of as an <i>enable</i> depite the ambiguity in the naming of the <i>Clearing</i> state.
<table> 
	<tr>
		<th> Previous State </th>
		<th> Transition In </th>
		<th> Transition Out </th>
		<th> Next State  </th> 
	</tr>
	<tr>
		<td> Stopped<b>-or-</b>Completed </td>
		<td> Reset Command </td> 
		<td> State Complete </td>
		<td> Idle </td> 
	</tr>
</table>
This method is called as required by <c>StateControl()</c>
</description> 

*)
CASE _MotorInitState OF
    0:
        IF _ComponentsReset = FALSE THEN
            _ComponentsReset := ResetOnResume();
        ELSE
            _MotorInitState := 1;
        END_IF

    1:
        IF _MotorsHomed = FALSE THEN
            _MotorsHomed := MotorsHome();
        ELSE
            _MotorInitState := 2;
        END_IF

    2:
        IF _MotorsReset = FALSE THEN
            _MotorsReset := MotorsInit();
        ELSE
            _MotorInitState := 3;

        END_IF

    3:
        IF _AlignNeeded THEN
            IF MotorsInitAlignGearIn() THEN
                _MotorInitState := 4;
            END_IF
        ELSE
            _MotorInitState := 4;
        END_IF

    4:
        SUPER^.Resetting();
END_CASE
END_METHOD

METHOD PROTECTED Starting
VAR_INPUT
END_VAR
IF ParseDone = FALSE THEN

    SUPER^.Starting();
ELSE

    SUPER^.Starting();
END_IF
END_METHOD

//! @summary This method contains code which will execute when this PackML module is in the <b>Suspending</b> state
METHOD PROTECTED Suspending
VAR
    i               : UDINT;
    SubModulesReady : BOOL := TRUE;
END_VAR

(*! <description><b>Note:</b> The <i>Suspend</i> command is intended to be initiated by automatic detection of upstream/downstream jams, etc. It is meant to be distinct from a <i>Hold</i> in that <i>Hold</i> should be commanded by an operator.  Both <i>Hold</i>and<i>Suspend</i> result in a <i>paused</i> state which should allow resumption of the <b>Execute</b> state. 
<table> 
	<tr>
		<th> Previous State </th>
		<th> Transition In </th>
		<th> Transition Out </th>
		<th> Next State  </th> 
	</tr>
	<tr>
		<td> Execute </td>
		<td> Suspend Command </td> 
		<td> State Complete </td>
		<td> Suspended </td> 
	</tr>
</table>
This method is called as required by <c>StateControl()</c>
</description> 

*)
_MotorsReset      := FALSE;
_MotorInitState   := 0;
_ComponentsReset  := FALSE;
_AlignGearInState := 0;
_Handshake_State  := 0;

SUPER^.Suspending();
END_METHOD

//! @summary This method contains code which will execute when this PackML module is in the <b>Unholding</b> state
METHOD PROTECTED Unholding
VAR
    i               : UDINT;
    SubModulesReady : BOOL := TRUE;
END_VAR

(*! <description><b></b><table> 
	<tr>
		<th> Previous State </th>
		<th> Transition In </th>
		<th> Transition Out </th>
		<th> Next State  </th> 
	</tr>
	<tr>
		<td> Held </td>
		<td> Unhold Command </td> 
		<td> State Complete </td>
		<td> Execute </td> 
	</tr>
</table>
This method is called as required by <c>StateControl()</c>
</description> 

*)
IF _ForceHold = FALSE THEN

    CASE _MotorInitState OF
        0:
            IF _ComponentsReset = FALSE THEN
                _ComponentsReset := ResetOnResume();
            ELSE
                _MotorInitState := 1;
            END_IF

        1:
            IF _MotorsHomed = FALSE THEN
                _MotorsHomed := MotorsHome();
            ELSE
                _MotorInitState := 2;
            END_IF

        2:
            IF _MotorsReset = FALSE THEN
                _MotorsReset := MotorsInit();
            ELSE
                _MotorInitState := 3;

            END_IF

        3:
            IF _AlignNeeded THEN
                IF MotorsInitAlignGearIn() THEN
                    _MotorInitState := 4;
                END_IF
            ELSE
                _MotorInitState := 4;
            END_IF

        4:
            FOR i := 1 TO NumberOfSubModules DO
                IF ipSubModules[i].CurrentState = E_PMLState.ePMLState_Held THEN
                    ipSubModules[i].StateCommand := ePMLCommand_Unhold;
                ELSIF ipSubModules[i].CurrentState = E_PMLState.ePMLState_Suspended THEN
                    ipSubModules[i].StateCommand := ePMLCommand_Unsuspend;
                END_IF
            END_FOR

            FOR i := 1 TO NumberOfSubModules DO
                SubModulesReady := SubModulesReady AND (ipSubModules[i].CurrentState = ePMLState_Execute);
            END_FOR

            IF SubModulesReady AND (StateTasksComplete OR NoStateTasksToComplete) THEN
                NoStateTasksToComplete := TRUE;
                StateTasksComplete     := FALSE;
                StateComplete();
            END_IF
    END_CASE

ELSE
    FOR i := 1 TO NumberOfSubModules DO
        IF ipSubModules[i].CurrentState = E_PMLState.ePMLState_Held THEN
            ipSubModules[i].StateCommand := ePMLCommand_Unhold;
        ELSIF ipSubModules[i].CurrentState = E_PMLState.ePMLState_Suspended THEN
            ipSubModules[i].StateCommand := ePMLCommand_Unsuspend;
        END_IF
    END_FOR

    FOR i := 1 TO NumberOfSubModules DO
        SubModulesReady := SubModulesReady AND (ipSubModules[i].CurrentState = ePMLState_Execute);
    END_FOR

    IF SubModulesReady AND (StateTasksComplete OR NoStateTasksToComplete) THEN
        NoStateTasksToComplete := TRUE;
        StateTasksComplete     := FALSE;
        StateComplete();
    END_IF
END_IF
END_METHOD

//! @summary This method contains code which will execute when this PackML module is in the <b>Unsuspending</b> state
METHOD PROTECTED Unsuspending
VAR
    i               : UDINT;
    SubModulesReady : BOOL := TRUE;
END_VAR

(*! <description><b></b><table> 
	<tr>
		<th> Previous State </th>
		<th> Transition In </th>
		<th> Transition Out </th>
		<th> Next State  </th> 
	</tr>
	<tr>
		<td> Suspended </td>
		<td> Unsuspend Command </td> 
		<td> State Complete </td>
		<td> Execute </td> 
	</tr>
</table>
This method is called as required by <c>StateControl()</c>
</description> 

*)
IF _ForceHold = FALSE THEN

    CASE _MotorInitState OF
        0:
            IF _ComponentsReset = FALSE THEN
                _ComponentsReset := ResetOnResume();
            ELSE
                _MotorInitState := 1;
            END_IF

        1:
            IF _MotorsHomed = FALSE THEN
                _MotorsHomed := MotorsHome();
            ELSE
                _MotorInitState := 2;
            END_IF

        2:
            IF _MotorsReset = FALSE THEN
                _MotorsReset := MotorsInit();
            ELSE
                _MotorInitState := 3;

            END_IF

        3:
            IF _AlignNeeded THEN
                IF MotorsInitAlignGearIn() THEN
                    _MotorInitState := 4;
                END_IF
            ELSE
                _MotorInitState := 4;
            END_IF

        4:
            SUPER^.Unsuspending();
    END_CASE

ELSE
    SUPER^.Unsuspending();
END_IF
END_METHOD

//! @summary This method serves as the entry point for all underlying FB logic

//! @description This method should be called cyclically by descendant function blocks by invoking <c>SUPER^.CyclicLogic()</c>.  Alternatively, the contents of this method could be reimplemented entirely in which case a call to this method would not be necessary.
METHOD PROTECTED Execute
VAR
    i : UDINT;
END_VAR
_MotorsReset := FALSE;

_MotorInitState := 0;

_ComponentsReset := FALSE;

// IF Global.AutoMode THEN

//     AutoSpeeds();

// ELSE

//     ManualSpeeds();

// END_IF

CASE _CurrentMode OF
    //=================================PRODUCTION MODE==================================
    E_PMLUnitMode.ePMLUnitMode_Production:
        ;

        //=================================MAINTENANCE MODE==================================	
    E_PMLUnitMode.ePMLUnitMode_Maintenance:
        ;

        //=================================MANUAL MODE==================================
    E_PMLUnitMode.ePMLUnitMode_Manual:
        ;

    E_PMLUnitMode.ePMLUnitMode_UserMode1:
        ;

END_CASE

// _MotorsInitialized := FALSE;

// _MotorsReset := FALSE;

SUPER^.Execute();
END_METHOD

METHOD PROTECTED Idle
VAR_INPUT
END_VAR
// ParseDone := FALSE;

// _MotorsReset := FALSE;

// _MotorInitState := 0;

// _ComponentsReset := FALSE;

// _AlignGearInState := 0;

// _Handshake_State := 0;

// 

// _CommandStates.Assembly_End_State := 0;

// _CommandStates.Assembly_Start_State := 0;

// _CommandStates.Generic_State := 0;

// _CommandStates.Nail_Lamination_State := 0;

// _CommandStates.Plate_State := 0;

// _CommandStates.SE_State := 0;

// _CommandStates.SENail_State := 0;

// _CommandStates.Stud_State := 0;

// _CommandStates.StudInfo_State := 0;

// _CommandStates.Wall_Info_State := 0;

// _CommandStates.MoveAborted := FALSE;

// _CommandStates.Last_Move_State := 0;

// _ExtractState := 0;

SUPER^.Idle();
END_METHOD

(*! @summary This method contains code which will execute when this PackML module is in the <b>Suspended</b> state*)
METHOD PROTECTED Suspended
// IF MessageBox_Data.ErrorPresent = FALSE AND AutoUnsuspendCheck_TON.Q AND AutoUnsuspendAvailable THEN
// 	ChangeState(State:=E_PMLCommand.ePMLCommand_Unsuspend);
// 	AutoUnsuspendAvailable := FALSE;
// END_IF
END_METHOD

PROPERTY CurrentStep : DINT
GET
CurrentStep := _CurrentStep;
END_GET
SET
_CurrentStep := CurrentStep;
END_SET
END_PROPERTY

PROPERTY EquipmentModuleID : E_EM_Index;
GET
EquipmentModuleID := _EquipmentModuleID;
END_GET
SET
_EquipmentModuleID := EquipmentModuleID;
END_SET
END_PROPERTY

PROPERTY ForceHold : Bool
GET
ForceHold := _ForceHold;
END_GET
SET
_ForceHold := ForceHold;
END_SET
END_PROPERTY

PROPERTY ParentResponseDefinitions : ARRAY[0..4] OF E_AlarmResponse
GET
ParentResponseDefinitions[TcEventSeverity.Verbose]  := E_AlarmResponse.NoResponse;
ParentResponseDefinitions[TcEventSeverity.Info]     := E_AlarmResponse.NoResponse;
ParentResponseDefinitions[TcEventSeverity.Warning]  := E_AlarmResponse.NoResponse;
ParentResponseDefinitions[TcEventSeverity.Error]    := E_AlarmResponse.Suspend_Controlled;
ParentResponseDefinitions[TcEventSeverity.Critical] := E_AlarmResponse.Suspend_Immediate;
END_GET
END_PROPERTY

PROPERTY RecoverBoardNum : DINT
SET
_RecoverBoardNum := RecoverBoardNum;
END_SET
END_PROPERTY

PROPERTY SafetyOK : BOOL
SET
_SafetyOK := SafetyOK;
END_SET
END_PROPERTY

PROPERTY TaskState : E_TaskState
GET
TaskState := _TaskState;
END_GET
SET
_TaskState := TaskState;
END_SET
END_PROPERTY

METHOD ClearAlarms
VAR_INPUT
    MyAlarms : ARRAY[1..Global.MAX_ALARM_COUNT] OF FB_TcAlarm;
END_VAR

VAR
    i : UDINT;
END_VAR
FOR i := 1 TO Global.MAX_ALARM_COUNT DO
    MyAlarms[i].Clear(0, 0);
END_FOR;
END_METHOD

METHOD ResetComponents : BOOL
VAR_INPUT
END_VAR
ResetComponents := TRUE;

FOR i := 1 TO NumberOfComponents DO
    ResetComponents := ipComponents[i].Reset() AND ResetComponents;
END_FOR

IF ResetComponents THEN
    _Error   := FALSE;
    _ErrorID := 0;
END_IF
END_METHOD

PROPERTY InSimulation : BOOL
SET
_InSimulation := InSimulation;
END_SET
END_PROPERTY

METHOD SimulationOff : BOOL
VAR_INPUT
END_VAR

VAR
    i : UDINT;
END_VAR
_InSimulation := FALSE;

// Call this module's subunits, if any are defined
FOR i := 1 TO NumberOfSubModules DO
    IF ipSubmodules_SR[i] <> 0 THEN
        ipSubModules_SR[i].SimulationOff();
    END_IF
END_FOR

FOR i := 1 TO NumberOfComponents DO
    ipComponents[i].InSimulation := FALSE;
END_FOR
END_METHOD

METHOD SimulationOn : BOOL
VAR_INPUT
END_VAR

VAR
    i : UDINT;

END_VAR
_InSimulation := TRUE;

// Call this module's subunits, if any are defined
FOR i := 1 TO NumberOfSubModules DO
    IF ipSubmodules_SR[i] <> 0 THEN
        ipSubModules_SR[i].SimulationOn();
    END_IF
END_FOR

FOR i := 1 TO NumberOfComponents DO
    IF ipComponents[i] <> 0 THEN
        ipComponents[i].InSimulation := TRUE;
    END_IF
END_FOR
END_METHOD

END_FUNCTION_BLOCK

// Machine/HMI Connections/FB_ControlSource_HMI
FUNCTION_BLOCK FB_ControlSource_HMI EXTENDS FB_CyclicFB IMPLEMENTS I_PackML_ExternalController
VAR_INPUT
    MainPMLControl_Simplified : ST_PackML_Control_Simplified;
END_VAR

VAR_OUTPUT
END_VAR

VAR
    ipModule                : I_PackML_Control;
    MainPMLControl_Standard : ST_PackML_Control;
    R_HMICommand            : R_TRIG;
END_VAR

METHOD CyclicLogic
VAR
    i : UDINT;
END_VAR
IF NOT _InitComplete THEN
    _InitComplete := Initialize();
    RETURN;
END_IF

MainPMLControl_Standard.CurrentMode  := ipModule.CurrentMode;
MainPMLControl_Standard.CurrentState := ipModule.CurrentState;

FOR i := 1 TO 5 DO
    MainPMLControl_Standard.ModeNames[i] := F_UnitModeToString(UDINT_TO_DINT(i));
END_FOR

//Process HMI requests
R_HMICommand(CLK := (MainPMLControl_Simplified.ResetPressed XOR
                    MainPMLControl_Simplified.StartPressed XOR
                    MainPMLControl_Simplified.HoldPressed XOR
                    MainPMLControl_Simplified.AbortPressed XOR
                    MainPMLControl_Simplified.StopPressed) XOR
                    (MainPMLControl_Standard.StateCommand <> E_PMLCommand.ePMLCommand_Undefined AND
                    ipModule.StateCommand <> MainPMLControl_Standard.StateCommand) XOR
                    (ipModule.ModeCommand <> MainPMLControl_Standard.ModeCommand));

